LIN {X 0,Y 566.425,Z 352.194,A -85,B 0,C 180,E1 -2599.455,E2 -2599.455} C_VEL
LIN {X 0,Y 566.296,Z 363.628,A -85,B 0,C 180,E1 -2600.355,E2 -2600.355} C_VEL
LIN {X 0,Y 566.162,Z 372.742,A -85,B 0,C 180,E1 -2601.254,E2 -2601.254} C_VEL
LIN {X 0,Y 566.096,Z 380.288,A -85,B 0,C 180,E1 -2602.151,E2 -2602.151} C_VEL
LIN {X 0,Y 566.007,Z 386.693,A -85,B 0,C 180,E1 -2603.065,E2 -2603.065} C_VEL
LIN {X 0,Y 565.99,Z 391.812,A -85,B 0,C 180,E1 -2603.942,E2 -2603.942} C_VEL
LIN {X 0,Y 565.878,Z 396.909,A -85,B 0,C 180,E1 -2605.013,E2 -2605.013} C_VEL
LIN {X 0,Y 565.927,Z 400.862,A -85,B 0,C 180,E1 -2606.084,E2 -2606.084} C_VEL
LIN {X 0,Y 565.878,Z 403.78,A -85,B 0,C 180,E1 -2607.153,E2 -2607.153} C_VEL
LIN {X 0,Y 565.846,Z 406.194,A -85,B 0,C 180,E1 -2608.577,E2 -2608.577} C_VEL
LIN {X 0,Y 565.841,Z 406.781,A -85,B 0,C 180,E1 -2609.288,E2 -2609.288} C_VEL
LIN {X 0,Y 565.841,Z 406.781,A -85,B 0,C 180,E1 -2610.712,E2 -2610.712} C_VEL
LIN {X 0,Y 565.846,Z 406.194,A -85,B 0,C 180,E1 -2611.423,E2 -2611.423} C_VEL
LIN {X 0,Y 565.878,Z 403.78,A -85,B 0,C 180,E1 -2612.847,E2 -2612.847} C_VEL
LIN {X 0,Y 565.927,Z 400.862,A -85,B 0,C 180,E1 -2613.916,E2 -2613.916} C_VEL
LIN {X 0,Y 565.878,Z 396.909,A -85,B 0,C 180,E1 -2614.987,E2 -2614.987} C_VEL
LIN {X 0,Y 565.991,Z 391.812,A -85,B 0,C 180,E1 -2616.058,E2 -2616.058} C_VEL
LIN {X 0,Y 566.035,Z 385.428,A -85,B 0,C 180,E1 -2617.132,E2 -2617.132} C_VEL
LIN {X 0,Y 566.134,Z 377.5,A -85,B 0,C 180,E1 -2618.207,E2 -2618.207} C_VEL
LIN {X 0,Y 566.239,Z 369.359,A -85,B 0,C 180,E1 -2619.105,E2 -2619.105} C_VEL
LIN {X 0,Y 566.339,Z 359.324,A -85,B 0,C 180,E1 -2620.005,E2 -2620.005} C_VEL
LIN {X 0,Y 566.458,Z 349.496,A -85,B 0,C 180,E1 -2620.725,E2 -2620.725} C_VEL
LIN {X 0,Y 566.565,Z 338.733,A -85,B 0,C 180,E1 -2621.366,E2 -2621.366} C_VEL
LIN {X 0,Y 566.736,Z 324.932,A -85,B 0,C 180,E1 -2621.988,E2 -2621.988} C_VEL
LIN {X 0,Y 566.892,Z 312.891,A -85,B 0,C 180,E1 -2622.371,E2 -2622.371} C_VEL
LIN {X 0,Y 566.7,Z 306.442,A -85,B 0,C 180,E1 -2622.534,E2 -2622.534} C_VEL
LIN {X 0,Y 565.903,Z 301.524,A -85,B 0,C 180,E1 -2622.643,E2 -2622.643} C_VEL
LIN {X 0,Y 565.956,Z 295.461,A -85,B 0,C 180,E1 -2625.116,E2 -2625.116} C_VEL
LIN {X 0,Y 566.005,Z 288.275,A -85,B 0,C 180,E1 -2628.084,E2 -2628.084} C_VEL
LIN {X 0,Y 566.01,Z 282.873,A -85,B 0,C 180,E1 -2630.344,E2 -2630.344} C_VEL
LIN {X 0,Y 566.031,Z 277.383,A -85,B 0,C 180,E1 -2632.637,E2 -2632.637} C_VEL
LIN {X 0,Y 566.079,Z 272.028,A -85,B 0,C 180,E1 -2634.997,E2 -2634.997} C_VEL
LIN {X 0,Y 566.145,Z 266.834,A -85,B 0,C 180,E1 -2637.342,E2 -2637.342} C_VEL
LIN {X 0,Y 566.199,Z 261.606,A -85,B 0,C 180,E1 -2639.768,E2 -2639.768} C_VEL
LIN {X 0,Y 566.325,Z 256.131,A -85,B 0,C 180,E1 -2642.447,E2 -2642.447} C_VEL
LIN {X 0,Y 566.395,Z 249.901,A -85,B 0,C 180,E1 -2645.674,E2 -2645.674} C_VEL
LIN {X 0,Y 566.483,Z 244.633,A -85,B 0,C 180,E1 -2648.59,E2 -2648.59} C_VEL
LIN {X 0,Y 566.516,Z 240.41,A -85,B 0,C 180,E1 -2651.108,E2 -2651.108} C_VEL
LIN {X 0,Y 566.447,Z 237.397,A -85,B 0,C 180,E1 -2653.03,E2 -2653.03} C_VEL
LIN {X 0,Y 566.232,Z 235.917,A -85,B 0,C 180,E1 -2654.031,E2 -2654.031} C_VEL
LIN {X 0,Y 566.168,Z 235.461,A -85,B 0,C 180,E1 -2655.035,E2 -2655.035} C_VEL
LIN {X 0,Y 566.176,Z 235.461,A -85,B 0,C 180,E1 -2657.907,E2 -2657.907} C_VEL
LIN {X 0,Y 566.209,Z 235.454,A -85,B 0,C 180,E1 -2660.723,E2 -2660.723} C_VEL
LIN {X 0,Y 566.181,Z 235.456,A -85,B 0,C 180,E1 -2663.426,E2 -2663.426} C_VEL
LIN {X 0,Y 566.213,Z 235.456,A -85,B 0,C 180,E1 -2666.264,E2 -2666.264} C_VEL
LIN {X 0,Y 566.185,Z 235.453,A -85,B 0,C 180,E1 -2668.922,E2 -2668.922} C_VEL
LIN {X 0,Y 566.188,Z 235.461,A -85,B 0,C 180,E1 -2671.853,E2 -2671.853} C_VEL
LIN {X 0,Y 566.238,Z 235.447,A -85,B 0,C 180,E1 -2675.036,E2 -2675.036} C_VEL
LIN {X 0,Y 566.189,Z 235.457,A -85,B 0,C 180,E1 -2678.134,E2 -2678.134} C_VEL
LIN {X 0,Y 566.228,Z 235.448,A -85,B 0,C 180,E1 -2680.611,E2 -2680.611} C_VEL
LIN {X 0,Y 566.194,Z 235.458,A -85,B 0,C 180,E1 -2683.408,E2 -2683.408} C_VEL
LIN {X 0,Y 566.183,Z 235.454,A -85,B 0,C 180,E1 -2686.355,E2 -2686.355} C_VEL
LIN {X 0,Y 566.226,Z 235.454,A -85,B 0,C 180,E1 -2689.267,E2 -2689.267} C_VEL
LIN {X 0,Y 566.179,Z 235.455,A -85,B 0,C 180,E1 -2692.148,E2 -2692.148} C_VEL
LIN {X 0,Y 566.231,Z 235.447,A -85,B 0,C 180,E1 -2694.298,E2 -2694.298} C_VEL
LIN {X 0,Y 566.255,Z 235.452,A -85,B 0,C 180,E1 -2697.15,E2 -2697.15} C_VEL
LIN {X 0,Y 566.265,Z 235.444,A -85,B 0,C 180,E1 -2699.996,E2 -2699.996} C_VEL
LIN {X 0,Y 566.25,Z 235.45,A -85,B 0,C 180,E1 -2702.841,E2 -2702.841} C_VEL
LIN {X 0,Y 566.235,Z 235.448,A -85,B 0,C 180,E1 -2705.694,E2 -2705.694} C_VEL
LIN {X 0,Y 566.178,Z 235.457,A -85,B 0,C 180,E1 -2708.562,E2 -2708.562} C_VEL
LIN {X 0,Y 566.231,Z 235.45,A -85,B 0,C 180,E1 -2711.45,E2 -2711.45} C_VEL
LIN {X 0,Y 566.205,Z 235.454,A -85,B 0,C 180,E1 -2714.5,E2 -2714.5} C_VEL
LIN {X 0,Y 566.171,Z 235.457,A -85,B 0,C 180,E1 -2717.327,E2 -2717.327} C_VEL
LIN {X 0,Y 566.19,Z 235.456,A -85,B 0,C 180,E1 -2720.332,E2 -2720.332} C_VEL
LIN {X 0,Y 566.141,Z 235.46,A -85,B 0,C 180,E1 -2723.277,E2 -2723.277} C_VEL
LIN {X 0,Y 566.178,Z 235.454,A -85,B 0,C 180,E1 -2725.744,E2 -2725.744} C_VEL
LIN {X 0,Y 566.178,Z 235.454,A -85,B 0,C 180,E1 -2727.457,E2 -2727.457} C_VEL
LIN {X 0,Y 565.499,Z 235.542,A -85,B 0,C 180,E1 -2728.051,E2 -2728.051} C_VEL
LIN {X 0,Y 562.63,Z 235.898,A -85,B 0,C 180,E1 -2729.015,E2 -2729.015} C_VEL
LIN {X 0,Y 560.214,Z 236.2,A -85,B 0,C 180,E1 -2729.79,E2 -2729.79} C_VEL
LIN {X 0,Y 559.183,Z 236.334,A -85,B 0,C 180,E1 -2730.389,E2 -2730.389} C_VEL
LIN {X 0,Y 559.102,Z 236.337,A -85,B 0,C 180,E1 -2730.592,E2 -2730.592} C_VEL
LIN {X 0,Y 559.137,Z 236.331,A -85,B 0,C 180,E1 -2733.569,E2 -2733.569} C_VEL
LIN {X 0,Y 559.146,Z 236.338,A -85,B 0,C 180,E1 -2736.447,E2 -2736.447} C_VEL
LIN {X 0,Y 559.131,Z 236.333,A -85,B 0,C 180,E1 -2738.929,E2 -2738.929} C_VEL
LIN {X 0,Y 559.154,Z 236.332,A -85,B 0,C 180,E1 -2741.762,E2 -2741.762} C_VEL
LIN {X 0,Y 559.109,Z 236.336,A -85,B 0,C 180,E1 -2744.733,E2 -2744.733} C_VEL
LIN {X 0,Y 559.134,Z 236.338,A -85,B 0,C 180,E1 -2747.857,E2 -2747.857} C_VEL
LIN {X 0,Y 559.14,Z 236.338,A -85,B 0,C 180,E1 -2750.132,E2 -2750.132} C_VEL
LIN {X 0,Y 559.091,Z 236.337,A -85,B 0,C 180,E1 -2752.889,E2 -2752.889} C_VEL
LIN {X 0,Y 559.105,Z 236.34,A -85,B 0,C 180,E1 -2755.553,E2 -2755.553} C_VEL
LIN {X 0,Y 559.118,Z 236.338,A -85,B 0,C 180,E1 -2758.135,E2 -2758.135} C_VEL
LIN {X 0,Y 559.12,Z 236.333,A -85,B 0,C 180,E1 -2760.646,E2 -2760.646} C_VEL
LIN {X 0,Y 559.12,Z 236.336,A -85,B 0,C 180,E1 -2763.167,E2 -2763.167} C_VEL
LIN {X 0,Y 559.11,Z 236.342,A -85,B 0,C 180,E1 -2765.493,E2 -2765.493} C_VEL
LIN {X 0,Y 559.104,Z 236.34,A -85,B 0,C 180,E1 -2767.846,E2 -2767.846} C_VEL
LIN {X 0,Y 559.131,Z 236.332,A -85,B 0,C 180,E1 -2770.49,E2 -2770.49} C_VEL
LIN {X 0,Y 559.146,Z 236.337,A -85,B 0,C 180,E1 -2773.197,E2 -2773.197} C_VEL
LIN {X 0,Y 559.12,Z 236.334,A -85,B 0,C 180,E1 -2776.183,E2 -2776.183} C_VEL
LIN {X 0,Y 559.171,Z 236.335,A -85,B 0,C 180,E1 -2779.133,E2 -2779.133} C_VEL
LIN {X 0,Y 559.149,Z 236.331,A -85,B 0,C 180,E1 -2782.053,E2 -2782.053} C_VEL
LIN {X 0,Y 559.203,Z 236.331,A -85,B 0,C 180,E1 -2784.953,E2 -2784.953} C_VEL
LIN {X 0,Y 559.183,Z 236.327,A -85,B 0,C 180,E1 -2787.839,E2 -2787.839} C_VEL
LIN {X 0,Y 559.219,Z 236.328,A -85,B 0,C 180,E1 -2790.72,E2 -2790.72} C_VEL
LIN {X 0,Y 559.187,Z 236.334,A -85,B 0,C 180,E1 -2792.882,E2 -2792.882} C_VEL
LIN {X 0,Y 559.173,Z 236.328,A -85,B 0,C 180,E1 -2795.771,E2 -2795.771} C_VEL
LIN {X 0,Y 559.149,Z 236.331,A -85,B 0,C 180,E1 -2797.947,E2 -2797.947} C_VEL
LIN {X 0,Y 559.171,Z 236.335,A -85,B 0,C 180,E1 -2800.867,E2 -2800.867} C_VEL
LIN {X 0,Y 559.12,Z 236.334,A -85,B 0,C 180,E1 -2803.817,E2 -2803.817} C_VEL
LIN {X 0,Y 559.146,Z 236.337,A -85,B 0,C 180,E1 -2806.803,E2 -2806.803} C_VEL
LIN {X 0,Y 559.113,Z 236.335,A -85,B 0,C 180,E1 -2809.839,E2 -2809.839} C_VEL
LIN {X 0,Y 559.103,Z 236.34,A -85,B 0,C 180,E1 -2812.154,E2 -2812.154} C_VEL
LIN {X 0,Y 559.11,Z 236.342,A -85,B 0,C 180,E1 -2814.507,E2 -2814.507} C_VEL
LIN {X 0,Y 559.118,Z 236.335,A -85,B 0,C 180,E1 -2816.904,E2 -2816.904} C_VEL
LIN {X 0,Y 559.141,Z 236.334,A -85,B 0,C 180,E1 -2819.871,E2 -2819.871} C_VEL
LIN {X 0,Y 559.118,Z 236.336,A -85,B 0,C 180,E1 -2822.717,E2 -2822.717} C_VEL
LIN {X 0,Y 559.101,Z 236.336,A -85,B 0,C 180,E1 -2825.325,E2 -2825.325} C_VEL
LIN {X 0,Y 559.09,Z 236.346,A -85,B 0,C 180,E1 -2828.02,E2 -2828.02} C_VEL
LIN {X 0,Y 559.125,Z 236.333,A -85,B 0,C 180,E1 -2830.814,E2 -2830.814} C_VEL
LIN {X 0,Y 559.111,Z 236.341,A -85,B 0,C 180,E1 -2833.736,E2 -2833.736} C_VEL
LIN {X 0,Y 559.129,Z 236.332,A -85,B 0,C 180,E1 -2836.804,E2 -2836.804} C_VEL
LIN {X 0,Y 559.132,Z 236.333,A -85,B 0,C 180,E1 -2839.194,E2 -2839.194} C_VEL
LIN {X 0,Y 559.09,Z 236.342,A -85,B 0,C 180,E1 -2841.987,E2 -2841.987} C_VEL
LIN {X 0,Y 559.116,Z 236.334,A -85,B 0,C 180,E1 -2844.683,E2 -2844.683} C_VEL
LIN {X 0,Y 559.135,Z 236.337,A -85,B 0,C 180,E1 -2847.366,E2 -2847.366} C_VEL
LIN {X 0,Y 559.111,Z 236.335,A -85,B 0,C 180,E1 -2850.147,E2 -2850.147} C_VEL
LIN {X 0,Y 559.136,Z 236.336,A -85,B 0,C 180,E1 -2853.102,E2 -2853.102} C_VEL
LIN {X 0,Y 559.124,Z 236.34,A -85,B 0,C 180,E1 -2855.5,E2 -2855.5} C_VEL
LIN {X 0,Y 559.147,Z 236.331,A -85,B 0,C 180,E1 -2858.629,E2 -2858.629} C_VEL
LIN {X 0,Y 559.14,Z 236.335,A -85,B 0,C 180,E1 -2860.931,E2 -2860.931} C_VEL
LIN {X 0,Y 559.139,Z 236.331,A -85,B 0,C 180,E1 -2863.952,E2 -2863.952} C_VEL
LIN {X 0,Y 559.144,Z 236.33,A -85,B 0,C 180,E1 -2866.189,E2 -2866.189} C_VEL
LIN {X 0,Y 559.186,Z 236.333,A -85,B 0,C 180,E1 -2869.138,E2 -2869.138} C_VEL
LIN {X 0,Y 559.173,Z 236.327,A -85,B 0,C 180,E1 -2872.058,E2 -2872.058} C_VEL
LIN {X 0,Y 559.231,Z 236.328,A -85,B 0,C 180,E1 -2874.958,E2 -2874.958} C_VEL
LIN {X 0,Y 559.223,Z 236.32,A -85,B 0,C 180,E1 -2877.844,E2 -2877.844} C_VEL
LIN {X 0,Y 559.267,Z 236.324,A -85,B 0,C 180,E1 -2880.724,E2 -2880.724} C_VEL
LIN {X 0,Y 559.22,Z 236.327,A -85,B 0,C 180,E1 -2882.886,E2 -2882.886} C_VEL
LIN {X 0,Y 559.202,Z 236.323,A -85,B 0,C 180,E1 -2885.774,E2 -2885.774} C_VEL
LIN {X 0,Y 559.154,Z 236.336,A -85,B 0,C 180,E1 -2888.679,E2 -2888.679} C_VEL
LIN {X 0,Y 559.196,Z 236.324,A -85,B 0,C 180,E1 -2891.604,E2 -2891.604} C_VEL
LIN {X 0,Y 559.197,Z 236.33,A -85,B 0,C 180,E1 -2894.599,E2 -2894.599} C_VEL
LIN {X 0,Y 559.129,Z 236.332,A -85,B 0,C 180,E1 -2897.561,E2 -2897.561} C_VEL
LIN {X 0,Y 559.161,Z 236.331,A -85,B 0,C 180,E1 -2899.841,E2 -2899.841} C_VEL
LIN {X 0,Y 559.137,Z 236.34,A -85,B 0,C 180,E1 -2902.156,E2 -2902.156} C_VEL
LIN {X 0,Y 559.154,Z 236.329,A -85,B 0,C 180,E1 -2905.302,E2 -2905.302} C_VEL
LIN {X 0,Y 559.128,Z 236.335,A -85,B 0,C 180,E1 -2908.534,E2 -2908.534} C_VEL
LIN {X 0,Y 559.142,Z 236.331,A -85,B 0,C 180,E1 -2911.275,E2 -2911.275} C_VEL
LIN {X 0,Y 559.166,Z 236.337,A -85,B 0,C 180,E1 -2913.951,E2 -2913.951} C_VEL
LIN {X 0,Y 559.131,Z 236.334,A -85,B 0,C 180,E1 -2917.112,E2 -2917.112} C_VEL
LIN {X 0,Y 559.16,Z 236.337,A -85,B 0,C 180,E1 -2919.943,E2 -2919.943} C_VEL
LIN {X 0,Y 559.149,Z 236.333,A -85,B 0,C 180,E1 -2922.747,E2 -2922.747} C_VEL
LIN {X 0,Y 559.128,Z 236.342,A -85,B 0,C 180,E1 -2925.261,E2 -2925.261} C_VEL
LIN {X 0,Y 559.491,Z 239.126,A -85,B 0,C 180,E1 -2927.289,E2 -2927.289} C_VEL
LIN {X 0,Y 559.518,Z 243.446,A -85,B 0,C 180,E1 -2930.017,E2 -2930.017} C_VEL
LIN {X 0,Y 559.416,Z 248.448,A -85,B 0,C 180,E1 -2932.914,E2 -2932.914} C_VEL
LIN {X 0,Y 559.316,Z 253.303,A -85,B 0,C 180,E1 -2935.568,E2 -2935.568} C_VEL
LIN {X 0,Y 559.244,Z 258.304,A -85,B 0,C 180,E1 -2938.143,E2 -2938.143} C_VEL
LIN {X 0,Y 559.118,Z 263.414,A -85,B 0,C 180,E1 -2940.646,E2 -2940.646} C_VEL
LIN {X 0,Y 559.095,Z 268.793,A -85,B 0,C 180,E1 -2943.19,E2 -2943.19} C_VEL
LIN {X 0,Y 558.976,Z 275.599,A -85,B 0,C 180,E1 -2946.276,E2 -2946.276} C_VEL
LIN {X 0,Y 558.99,Z 280.952,A -85,B 0,C 180,E1 -2948.617,E2 -2948.617} C_VEL
LIN {X 0,Y 558.923,Z 288.261,A -85,B 0,C 180,E1 -2951.679,E2 -2951.679} C_VEL
LIN {X 0,Y 558.869,Z 295.461,A -85,B 0,C 180,E1 -2954.688,E2 -2954.688} C_VEL
LIN {X 0,Y 558.838,Z 301.524,A -85,B 0,C 180,E1 -2957.194,E2 -2957.194} C_VEL
LIN {X 0,Y 559.997,Z 310.238,A -85,B 0,C 180,E1 -2957.405,E2 -2957.405} C_VEL
LIN {X 0,Y 559.848,Z 321.177,A -85,B 0,C 180,E1 -2957.729,E2 -2957.729} C_VEL
LIN {X 0,Y 559.718,Z 330.187,A -85,B 0,C 180,E1 -2958.08,E2 -2958.08} C_VEL
LIN {X 0,Y 559.585,Z 340.522,A -85,B 0,C 180,E1 -2958.592,E2 -2958.592} C_VEL
LIN {X 0,Y 559.46,Z 350.83,A -85,B 0,C 180,E1 -2959.231,E2 -2959.231} C_VEL
LIN {X 0,Y 559.317,Z 360.442,A -85,B 0,C 180,E1 -2959.96,E2 -2959.96} C_VEL
LIN {X 0,Y 559.197,Z 371.11,A -85,B 0,C 180,E1 -2960.962,E2 -2960.962} C_VEL
LIN {X 0,Y 559.051,Z 378.909,A -85,B 0,C 180,E1 -2961.87,E2 -2961.87} C_VEL
LIN {X 0,Y 558.977,Z 385.419,A -85,B 0,C 180,E1 -2962.777,E2 -2962.777} C_VEL
LIN {X 0,Y 558.91,Z 391.803,A -85,B 0,C 180,E1 -2963.864,E2 -2963.864} C_VEL
LIN {X 0,Y 558.798,Z 396.9,A -85,B 0,C 180,E1 -2964.949,E2 -2964.949} C_VEL
LIN {X 0,Y 558.845,Z 400.855,A -85,B 0,C 180,E1 -2966.034,E2 -2966.034} C_VEL
LIN {X 0,Y 558.8,Z 403.775,A -85,B 0,C 180,E1 -2967.116,E2 -2967.116} C_VEL
LIN {X 0,Y 558.745,Z 406.195,A -85,B 0,C 180,E1 -2968.559,E2 -2968.559} C_VEL
LIN {X 0,Y 558.741,Z 406.78,A -85,B 0,C 180,E1 -2969.279,E2 -2969.279} C_VEL
LIN {X 0,Y 558.741,Z 406.78,A -85,B 0,C 180,E1 -2970.721,E2 -2970.721} C_VEL
LIN {X 0,Y 558.745,Z 406.195,A -85,B 0,C 180,E1 -2971.441,E2 -2971.441} C_VEL
LIN {X 0,Y 558.8,Z 403.775,A -85,B 0,C 180,E1 -2972.884,E2 -2972.884} C_VEL
LIN {X 0,Y 558.845,Z 400.855,A -85,B 0,C 180,E1 -2973.966,E2 -2973.966} C_VEL
LIN {X 0,Y 558.798,Z 396.9,A -85,B 0,C 180,E1 -2975.051,E2 -2975.051} C_VEL
LIN {X 0,Y 558.911,Z 391.803,A -85,B 0,C 180,E1 -2976.136,E2 -2976.136} C_VEL
LIN {X 0,Y 558.977,Z 385.419,A -85,B 0,C 180,E1 -2977.223,E2 -2977.223} C_VEL
LIN {X 0,Y 559.098,Z 377.503,A -85,B 0,C 180,E1 -2978.311,E2 -2978.311} C_VEL
LIN {X 0,Y 559.212,Z 369.36,A -85,B 0,C 180,E1 -2979.22,E2 -2979.22} C_VEL
LIN {X 0,Y 559.349,Z 359.311,A -85,B 0,C 180,E1 -2980.131,E2 -2980.131} C_VEL
LIN {X 0,Y 559.46,Z 350.83,A -85,B 0,C 180,E1 -2980.769,E2 -2980.769} C_VEL
LIN {X 0,Y 559.578,Z 340.587,A -85,B 0,C 180,E1 -2981.404,E2 -2981.404} C_VEL
LIN {X 0,Y 559.729,Z 330.496,A -85,B 0,C 180,E1 -2981.906,E2 -2981.906} C_VEL
LIN {X 0,Y 559.875,Z 319.762,A -85,B 0,C 180,E1 -2982.321,E2 -2982.321} C_VEL
LIN {X 0,Y 559.823,Z 307.537,A -85,B 0,C 180,E1 -2982.668,E2 -2982.668} C_VEL
LIN {X 0,Y 558.839,Z 301.524,A -85,B 0,C 180,E1 -2982.806,E2 -2982.806} C_VEL
LIN {X 0,Y 558.869,Z 295.461,A -85,B 0,C 180,E1 -2985.312,E2 -2985.312} C_VEL
LIN {X 0,Y 558.923,Z 288.261,A -85,B 0,C 180,E1 -2988.321,E2 -2988.321} C_VEL
LIN {X 0,Y 558.99,Z 280.952,A -85,B 0,C 180,E1 -2991.383,E2 -2991.383} C_VEL
LIN {X 0,Y 558.998,Z 273.846,A -85,B 0,C 180,E1 -2994.512,E2 -2994.512} C_VEL
LIN {X 0,Y 559.077,Z 268.585,A -85,B 0,C 180,E1 -2996.906,E2 -2996.906} C_VEL
LIN {X 0,Y 559.17,Z 262.314,A -85,B 0,C 180,E1 -2999.859,E2 -2999.859} C_VEL
LIN {X 0,Y 559.281,Z 256.61,A -85,B 0,C 180,E1 -3002.706,E2 -3002.706} C_VEL
LIN {X 0,Y 559.387,Z 251.651,A -85,B 0,C 180,E1 -3005.304,E2 -3005.304} C_VEL
LIN {X 0,Y 559.435,Z 246.829,A -85,B 0,C 180,E1 -3007.992,E2 -3007.992} C_VEL
LIN {X 0,Y 559.522,Z 242.141,A -85,B 0,C 180,E1 -3010.779,E2 -3010.779} C_VEL
LIN {X 0,Y 559.411,Z 238.339,A -85,B 0,C 180,E1 -3013.223,E2 -3013.223} C_VEL
LIN {X 0,Y 559.125,Z 236.341,A -85,B 0,C 180,E1 -3014.739,E2 -3014.739} C_VEL
LIN {X 0,Y 559.144,Z 236.337,A -85,B 0,C 180,E1 -3017.865,E2 -3017.865} C_VEL
LIN {X 0,Y 559.178,Z 236.335,A -85,B 0,C 180,E1 -3020.132,E2 -3020.132} C_VEL
LIN {X 0,Y 559.131,Z 236.334,A -85,B 0,C 180,E1 -3022.888,E2 -3022.888} C_VEL
LIN {X 0,Y 559.166,Z 236.337,A -85,B 0,C 180,E1 -3026.049,E2 -3026.049} C_VEL
LIN {X 0,Y 559.15,Z 236.329,A -85,B 0,C 180,E1 -3028.978,E2 -3028.978} C_VEL
LIN {X 0,Y 559.134,Z 236.336,A -85,B 0,C 180,E1 -3031.623,E2 -3031.623} C_VEL
LIN {X 0,Y 559.161,Z 236.328,A -85,B 0,C 180,E1 -3034.814,E2 -3034.814} C_VEL
LIN {X 0,Y 559.137,Z 236.34,A -85,B 0,C 180,E1 -3037.844,E2 -3037.844} C_VEL
LIN {X 0,Y 559.19,Z 236.325,A -85,B 0,C 180,E1 -3040.491,E2 -3040.491} C_VEL
LIN {X 0,Y 559.162,Z 236.331,A -85,B 0,C 180,E1 -3043.194,E2 -3043.194} C_VEL
LIN {X 0,Y 559.16,Z 236.33,A -85,B 0,C 180,E1 -3046.18,E2 -3046.18} C_VEL
LIN {X 0,Y 559.184,Z 236.329,A -85,B 0,C 180,E1 -3049.13,E2 -3049.13} C_VEL
LIN {X 0,Y 559.133,Z 236.333,A -85,B 0,C 180,E1 -3052.049,E2 -3052.049} C_VEL
LIN {X 0,Y 559.202,Z 236.323,A -85,B 0,C 180,E1 -3054.226,E2 -3054.226} C_VEL
LIN {X 0,Y 559.22,Z 236.327,A -85,B 0,C 180,E1 -3057.114,E2 -3057.114} C_VEL
LIN {X 0,Y 559.237,Z 236.319,A -85,B 0,C 180,E1 -3059.996,E2 -3059.996} C_VEL
LIN {X 0,Y 559.218,Z 236.326,A -85,B 0,C 180,E1 -3062.877,E2 -3062.877} C_VEL
LIN {X 0,Y 559.202,Z 236.324,A -85,B 0,C 180,E1 -3065.766,E2 -3065.766} C_VEL
LIN {X 0,Y 559.144,Z 236.334,A -85,B 0,C 180,E1 -3068.67,E2 -3068.67} C_VEL
LIN {X 0,Y 559.188,Z 236.326,A -85,B 0,C 180,E1 -3071.596,E2 -3071.596} C_VEL
LIN {X 0,Y 559.176,Z 236.331,A -85,B 0,C 180,E1 -3074.591,E2 -3074.591} C_VEL
LIN {X 0,Y 559.115,Z 236.334,A -85,B 0,C 180,E1 -3077.553,E2 -3077.553} C_VEL
LIN {X 0,Y 559.146,Z 236.33,A -85,B 0,C 180,E1 -3079.833,E2 -3079.833} C_VEL
LIN {X 0,Y 559.111,Z 236.336,A -85,B 0,C 180,E1 -3082.148,E2 -3082.148} C_VEL
LIN {X 0,Y 559.142,Z 236.331,A -85,B 0,C 180,E1 -3085.293,E2 -3085.293} C_VEL
LIN {X 0,Y 559.137,Z 236.338,A -85,B 0,C 180,E1 -3088.378,E2 -3088.378} C_VEL
LIN {X 0,Y 559.102,Z 236.337,A -85,B 0,C 180,E1 -3090.592,E2 -3090.592} C_VEL
LIN {X 0,Y 558.44,Z 236.42,A -85,B 0,C 180,E1 -3091.193,E2 -3091.193} C_VEL
LIN {X 0,Y 555.583,Z 236.779,A -85,B 0,C 180,E1 -3092.169,E2 -3092.169} C_VEL
LIN {X 0,Y 553.175,Z 237.076,A -85,B 0,C 180,E1 -3092.955,E2 -3092.955} C_VEL
LIN {X 0,Y 552.156,Z 237.201,A -85,B 0,C 180,E1 -3093.562,E2 -3093.562} C_VEL
LIN {X 0,Y 552.082,Z 237.211,A -85,B 0,C 180,E1 -3093.767,E2 -3093.767} C_VEL
LIN {X 0,Y 552.074,Z 237.214,A -85,B 0,C 180,E1 -3096.742,E2 -3096.742} C_VEL
LIN {X 0,Y 552.088,Z 237.21,A -85,B 0,C 180,E1 -3099.522,E2 -3099.522} C_VEL
LIN {X 0,Y 552.124,Z 237.205,A -85,B 0,C 180,E1 -3101.437,E2 -3101.437} C_VEL
LIN {X 0,Y 552.067,Z 237.215,A -85,B 0,C 180,E1 -3104.53,E2 -3104.53} C_VEL
LIN {X 0,Y 552.078,Z 237.213,A -85,B 0,C 180,E1 -3107.58,E2 -3107.58} C_VEL
LIN {X 0,Y 552.102,Z 237.21,A -85,B 0,C 180,E1 -3110.472,E2 -3110.472} C_VEL
LIN {X 0,Y 552.057,Z 237.215,A -85,B 0,C 180,E1 -3113.312,E2 -3113.312} C_VEL
LIN {X 0,Y 552.082,Z 237.218,A -85,B 0,C 180,E1 -3115.937,E2 -3115.937} C_VEL
LIN {X 0,Y 552.057,Z 237.214,A -85,B 0,C 180,E1 -3118.537,E2 -3118.537} C_VEL
LIN {X 0,Y 552.083,Z 237.215,A -85,B 0,C 180,E1 -3121.431,E2 -3121.431} C_VEL
LIN {X 0,Y 552.11,Z 237.207,A -85,B 0,C 180,E1 -3124.355,E2 -3124.355} C_VEL
LIN {X 0,Y 552.092,Z 237.209,A -85,B 0,C 180,E1 -3126.758,E2 -3126.758} C_VEL
LIN {X 0,Y 552.072,Z 237.215,A -85,B 0,C 180,E1 -3129.897,E2 -3129.897} C_VEL
LIN {X 0,Y 552.125,Z 237.209,A -85,B 0,C 180,E1 -3132.977,E2 -3132.977} C_VEL
LIN {X 0,Y 552.078,Z 237.213,A -85,B 0,C 180,E1 -3136.003,E2 -3136.003} C_VEL
LIN {X 0,Y 552.129,Z 237.21,A -85,B 0,C 180,E1 -3138.993,E2 -3138.993} C_VEL
LIN {X 0,Y 552.103,Z 237.209,A -85,B 0,C 180,E1 -3141.951,E2 -3141.951} C_VEL
LIN {X 0,Y 552.143,Z 237.204,A -85,B 0,C 180,E1 -3144.156,E2 -3144.156} C_VEL
LIN {X 0,Y 552.153,Z 237.21,A -85,B 0,C 180,E1 -3147.082,E2 -3147.082} C_VEL
LIN {X 0,Y 552.158,Z 237.202,A -85,B 0,C 180,E1 -3150,E2 -3150} C_VEL
LIN {X 0,Y 552.153,Z 237.21,A -85,B 0,C 180,E1 -3152.918,E2 -3152.918} C_VEL
LIN {X 0,Y 552.143,Z 237.204,A -85,B 0,C 180,E1 -3155.844,E2 -3155.844} C_VEL
LIN {X 0,Y 552.103,Z 237.209,A -85,B 0,C 180,E1 -3158.049,E2 -3158.049} C_VEL
LIN {X 0,Y 552.129,Z 237.21,A -85,B 0,C 180,E1 -3161.007,E2 -3161.007} C_VEL
LIN {X 0,Y 552.078,Z 237.213,A -85,B 0,C 180,E1 -3163.997,E2 -3163.997} C_VEL
LIN {X 0,Y 552.126,Z 237.206,A -85,B 0,C 180,E1 -3167.343,E2 -3167.343} C_VEL
LIN {X 0,Y 552.072,Z 237.215,A -85,B 0,C 180,E1 -3170.103,E2 -3170.103} C_VEL
LIN {X 0,Y 552.092,Z 237.209,A -85,B 0,C 180,E1 -3173.242,E2 -3173.242} C_VEL
LIN {X 0,Y 552.11,Z 237.207,A -85,B 0,C 180,E1 -3175.645,E2 -3175.645} C_VEL
LIN {X 0,Y 552.083,Z 237.215,A -85,B 0,C 180,E1 -3178.569,E2 -3178.569} C_VEL
LIN {X 0,Y 552.074,Z 237.212,A -85,B 0,C 180,E1 -3181.483,E2 -3181.483} C_VEL
LIN {X 0,Y 552.088,Z 237.219,A -85,B 0,C 180,E1 -3184.176,E2 -3184.176} C_VEL
LIN {X 0,Y 552.055,Z 237.214,A -85,B 0,C 180,E1 -3186.75,E2 -3186.75} C_VEL
LIN {X 0,Y 552.114,Z 237.208,A -85,B 0,C 180,E1 -3189.527,E2 -3189.527} C_VEL
LIN {X 0,Y 552.078,Z 237.213,A -85,B 0,C 180,E1 -3192.429,E2 -3192.429} C_VEL
LIN {X 0,Y 552.071,Z 237.216,A -85,B 0,C 180,E1 -3195.569,E2 -3195.569} C_VEL
LIN {X 0,Y 552.124,Z 237.205,A -85,B 0,C 180,E1 -3198.677,E2 -3198.677} C_VEL
LIN {X 0,Y 552.074,Z 237.216,A -85,B 0,C 180,E1 -3201.416,E2 -3201.416} C_VEL
LIN {X 0,Y 552.07,Z 237.214,A -85,B 0,C 180,E1 -3204.163,E2 -3204.163} C_VEL
LIN {X 0,Y 552.089,Z 237.209,A -85,B 0,C 180,E1 -3206.82,E2 -3206.82} C_VEL
LIN {X 0,Y 552.065,Z 237.22,A -85,B 0,C 180,E1 -3209.395,E2 -3209.395} C_VEL
LIN {X 0,Y 552.091,Z 237.212,A -85,B 0,C 180,E1 -3211.907,E2 -3211.907} C_VEL
LIN {X 0,Y 552.122,Z 237.206,A -85,B 0,C 180,E1 -3214.654,E2 -3214.654} C_VEL
LIN {X 0,Y 552.062,Z 237.218,A -85,B 0,C 180,E1 -3217.554,E2 -3217.554} C_VEL
LIN {X 0,Y 552.122,Z 237.205,A -85,B 0,C 180,E1 -3220.378,E2 -3220.378} C_VEL
LIN {X 0,Y 552.129,Z 237.21,A -85,B 0,C 180,E1 -3222.982,E2 -3222.982} C_VEL
LIN {X 0,Y 552.109,Z 237.207,A -85,B 0,C 180,E1 -3226.009,E2 -3226.009} C_VEL
LIN {X 0,Y 552.155,Z 237.21,A -85,B 0,C 180,E1 -3228.998,E2 -3228.998} C_VEL
LIN {X 0,Y 552.128,Z 237.204,A -85,B 0,C 180,E1 -3231.956,E2 -3231.956} C_VEL
LIN {X 0,Y 552.206,Z 237.204,A -85,B 0,C 180,E1 -3234.893,E2 -3234.893} C_VEL
LIN {X 0,Y 552.197,Z 237.196,A -85,B 0,C 180,E1 -3237.816,E2 -3237.816} C_VEL
LIN {X 0,Y 552.236,Z 237.2,A -85,B 0,C 180,E1 -3240.733,E2 -3240.733} C_VEL
LIN {X 0,Y 552.185,Z 237.203,A -85,B 0,C 180,E1 -3242.922,E2 -3242.922} C_VEL
LIN {X 0,Y 552.175,Z 237.199,A -85,B 0,C 180,E1 -3245.848,E2 -3245.848} C_VEL
LIN {X 0,Y 552.127,Z 237.21,A -85,B 0,C 180,E1 -3248.79,E2 -3248.79} C_VEL
LIN {X 0,Y 552.152,Z 237.202,A -85,B 0,C 180,E1 -3251.754,E2 -3251.754} C_VEL
LIN {X 0,Y 552.132,Z 237.208,A -85,B 0,C 180,E1 -3254.752,E2 -3254.752} C_VEL
LIN {X 0,Y 552.088,Z 237.211,A -85,B 0,C 180,E1 -3257.793,E2 -3257.793} C_VEL
LIN {X 0,Y 552.122,Z 237.212,A -85,B 0,C 180,E1 -3260.105,E2 -3260.105} C_VEL
LIN {X 0,Y 552.088,Z 237.215,A -85,B 0,C 180,E1 -3262.454,E2 -3262.454} C_VEL
LIN {X 0,Y 552.121,Z 237.205,A -85,B 0,C 180,E1 -3265.346,E2 -3265.346} C_VEL
LIN {X 0,Y 552.095,Z 237.211,A -85,B 0,C 180,E1 -3268.559,E2 -3268.559} C_VEL
LIN {X 0,Y 552.114,Z 237.208,A -85,B 0,C 180,E1 -3271.478,E2 -3271.478} C_VEL
LIN {X 0,Y 552.107,Z 237.213,A -85,B 0,C 180,E1 -3274.168,E2 -3274.168} C_VEL
LIN {X 0,Y 552.1,Z 237.209,A -85,B 0,C 180,E1 -3276.75,E2 -3276.75} C_VEL
LIN {X 0,Y 552.129,Z 237.212,A -85,B 0,C 180,E1 -3279.53,E2 -3279.53} C_VEL
LIN {X 0,Y 552.112,Z 237.211,A -85,B 0,C 180,E1 -3282.43,E2 -3282.43} C_VEL
LIN {X 0,Y 552.085,Z 237.216,A -85,B 0,C 180,E1 -3284.532,E2 -3284.532} C_VEL
LIN {X 0,Y 552.165,Z 237.846,A -85,B 0,C 180,E1 -3285.571,E2 -3285.571} C_VEL
LIN {X 0,Y 552.511,Z 240.819,A -85,B 0,C 180,E1 -3287.612,E2 -3287.612} C_VEL
LIN {X 0,Y 552.485,Z 245.424,A -85,B 0,C 180,E1 -3290.504,E2 -3290.504} C_VEL
LIN {X 0,Y 552.408,Z 250.167,A -85,B 0,C 180,E1 -3293.277,E2 -3293.277} C_VEL
LIN {X 0,Y 552.289,Z 255.054,A -85,B 0,C 180,E1 -3295.951,E2 -3295.951} C_VEL
LIN {X 0,Y 552.164,Z 260.043,A -85,B 0,C 180,E1 -3298.544,E2 -3298.544} C_VEL
LIN {X 0,Y 552.074,Z 265.941,A -85,B 0,C 180,E1 -3301.45,E2 -3301.45} C_VEL
LIN {X 0,Y 551.961,Z 272.09,A -85,B 0,C 180,E1 -3304.348,E2 -3304.348} C_VEL
LIN {X 0,Y 551.907,Z 277.35,A -85,B 0,C 180,E1 -3306.75,E2 -3306.75} C_VEL
LIN {X 0,Y 551.865,Z 282.689,A -85,B 0,C 180,E1 -3309.11,E2 -3309.11} C_VEL
LIN {X 0,Y 551.839,Z 288.17,A -85,B 0,C 180,E1 -3311.435,E2 -3311.435} C_VEL
LIN {X 0,Y 551.784,Z 293.639,A -85,B 0,C 180,E1 -3313.728,E2 -3313.728} C_VEL
LIN {X 0,Y 551.762,Z 299.054,A -85,B 0,C 180,E1 -3315.995,E2 -3315.995} C_VEL
LIN {X 0,Y 551.736,Z 301.524,A -85,B 0,C 180,E1 -3317.026,E2 -3317.026} C_VEL
LIN {X 0,Y 553.043,Z 310.206,A -85,B 0,C 180,E1 -3317.244,E2 -3317.244} C_VEL
LIN {X 0,Y 552.926,Z 321.029,A -85,B 0,C 180,E1 -3317.568,E2 -3317.568} C_VEL
LIN {X 0,Y 552.752,Z 331.375,A -85,B 0,C 180,E1 -3317.983,E2 -3317.983} C_VEL
LIN {X 0,Y 552.595,Z 341.456,A -85,B 0,C 180,E1 -3318.5,E2 -3318.5} C_VEL
LIN {X 0,Y 552.47,Z 350.814,A -85,B 0,C 180,E1 -3319.093,E2 -3319.093} C_VEL
LIN {X 0,Y 552.301,Z 360.43,A -85,B 0,C 180,E1 -3319.831,E2 -3319.831} C_VEL
LIN {X 0,Y 552.152,Z 371.103,A -85,B 0,C 180,E1 -3320.845,E2 -3320.845} C_VEL
LIN {X 0,Y 552.014,Z 378.901,A -85,B 0,C 180,E1 -3321.765,E2 -3321.765} C_VEL
LIN {X 0,Y 551.907,Z 385.41,A -85,B 0,C 180,E1 -3322.684,E2 -3322.684} C_VEL
LIN {X 0,Y 551.812,Z 391.107,A -85,B 0,C 180,E1 -3323.653,E2 -3323.653} C_VEL
LIN {X 0,Y 551.803,Z 395.348,A -85,B 0,C 180,E1 -3324.519,E2 -3324.519} C_VEL
LIN {X 0,Y 551.767,Z 399.64,A -85,B 0,C 180,E1 -3325.617,E2 -3325.617} C_VEL
LIN {X 0,Y 551.751,Z 401.976,A -85,B 0,C 180,E1 -3326.349,E2 -3326.349} C_VEL
LIN {X 0,Y 551.724,Z 403.77,A -85,B 0,C 180,E1 -3327.079,E2 -3327.079} C_VEL
LIN {X 0,Y 551.645,Z 406.195,A -85,B 0,C 180,E1 -3328.54,E2 -3328.54} C_VEL
LIN {X 0,Y 551.641,Z 406.78,A -85,B 0,C 180,E1 -3329.27,E2 -3329.27} C_VEL
LIN {X 0,Y 551.641,Z 406.78,A -85,B 0,C 180,E1 -3330.73,E2 -3330.73} C_VEL
LIN {X 0,Y 551.645,Z 406.195,A -85,B 0,C 180,E1 -3331.46,E2 -3331.46} C_VEL
LIN {X 0,Y 551.724,Z 403.77,A -85,B 0,C 180,E1 -3332.921,E2 -3332.921} C_VEL
LIN {X 0,Y 551.765,Z 400.848,A -85,B 0,C 180,E1 -3334.017,E2 -3334.017} C_VEL
LIN {X 0,Y 551.724,Z 396.892,A -85,B 0,C 180,E1 -3335.116,E2 -3335.116} C_VEL
LIN {X 0,Y 551.838,Z 392.402,A -85,B 0,C 180,E1 -3336.097,E2 -3336.097} C_VEL
LIN {X 0,Y 551.89,Z 386.56,A -85,B 0,C 180,E1 -3337.132,E2 -3337.132} C_VEL
LIN {X 0,Y 551.986,Z 380.271,A -85,B 0,C 180,E1 -3338.051,E2 -3338.051} C_VEL
LIN {X 0,Y 552.124,Z 372.725,A -85,B 0,C 180,E1 -3338.971,E2 -3338.971} C_VEL
LIN {X 0,Y 552.274,Z 363.618,A -85,B 0,C 180,E1 -3339.892,E2 -3339.892} C_VEL
LIN {X 0,Y 552.45,Z 352.163,A -85,B 0,C 180,E1 -3340.815,E2 -3340.815} C_VEL
LIN {X 0,Y 552.571,Z 343.467,A -85,B 0,C 180,E1 -3341.386,E2 -3341.386} C_VEL
LIN {X 0,Y 552.745,Z 333.386,A -85,B 0,C 180,E1 -3341.924,E2 -3341.924} C_VEL
LIN {X 0,Y 552.892,Z 323.602,A -85,B 0,C 180,E1 -3342.34,E2 -3342.34} C_VEL
LIN {X 0,Y 553.04,Z 312.827,A -85,B 0,C 180,E1 -3342.686,E2 -3342.686} C_VEL
LIN {X 0,Y 552.767,Z 307.533,A -85,B 0,C 180,E1 -3342.832,E2 -3342.832} C_VEL
LIN {X 0,Y 551.737,Z 301.524,A -85,B 0,C 180,E1 -3342.974,E2 -3342.974} C_VEL
LIN {X 0,Y 551.783,Z 295.46,A -85,B 0,C 180,E1 -3345.514,E2 -3345.514} C_VEL
LIN {X 0,Y 551.839,Z 289.995,A -85,B 0,C 180,E1 -3347.797,E2 -3347.797} C_VEL
LIN {X 0,Y 551.852,Z 284.517,A -85,B 0,C 180,E1 -3350.111,E2 -3350.111} C_VEL
LIN {X 0,Y 551.885,Z 279.104,A -85,B 0,C 180,E1 -3352.459,E2 -3352.459} C_VEL
LIN {X 0,Y 551.946,Z 272.851,A -85,B 0,C 180,E1 -3355.302,E2 -3355.302} C_VEL
LIN {X 0,Y 552.037,Z 266.84,A -85,B 0,C 180,E1 -3358.102,E2 -3358.102} C_VEL
LIN {X 0,Y 552.12,Z 261.722,A -85,B 0,C 180,E1 -3360.607,E2 -3360.607} C_VEL
LIN {X 0,Y 552.245,Z 256.688,A -85,B 0,C 180,E1 -3363.176,E2 -3363.176} C_VEL
LIN {X 0,Y 552.357,Z 251.767,A -85,B 0,C 180,E1 -3365.822,E2 -3365.822} C_VEL
LIN {X 0,Y 552.446,Z 246.976,A -85,B 0,C 180,E1 -3368.561,E2 -3368.561} C_VEL
LIN {X 0,Y 552.51,Z 243.834,A -85,B 0,C 180,E1 -3370.444,E2 -3370.444} C_VEL
LIN {X 0,Y 552.511,Z 240.689,A -85,B 0,C 180,E1 -3372.456,E2 -3372.456} C_VEL
LIN {X 0,Y 552.137,Z 237.7,A -85,B 0,C 180,E1 -3374.534,E2 -3374.534} C_VEL
LIN {X 0,Y 552.086,Z 237.216,A -85,B 0,C 180,E1 -3375.559,E2 -3375.559} C_VEL
LIN {X 0,Y 552.11,Z 237.212,A -85,B 0,C 180,E1 -3378.678,E2 -3378.678} C_VEL
LIN {X 0,Y 552.115,Z 237.208,A -85,B 0,C 180,E1 -3381.408,E2 -3381.408} C_VEL
LIN {X 0,Y 552.073,Z 237.221,A -85,B 0,C 180,E1 -3384.153,E2 -3384.153} C_VEL
LIN {X 0,Y 552.115,Z 237.206,A -85,B 0,C 180,E1 -3386.811,E2 -3386.811} C_VEL
LIN {X 0,Y 552.094,Z 237.21,A -85,B 0,C 180,E1 -3389.387,E2 -3389.387} C_VEL
LIN {X 0,Y 552.077,Z 237.22,A -85,B 0,C 180,E1 -3391.897,E2 -3391.897} C_VEL
LIN {X 0,Y 552.121,Z 237.205,A -85,B 0,C 180,E1 -3394.654,E2 -3394.654} C_VEL
LIN {X 0,Y 552.088,Z 237.215,A -85,B 0,C 180,E1 -3397.546,E2 -3397.546} C_VEL
LIN {X 0,Y 552.142,Z 237.204,A -85,B 0,C 180,E1 -3400.372,E2 -3400.372} C_VEL
LIN {X 0,Y 552.118,Z 237.206,A -85,B 0,C 180,E1 -3402.973,E2 -3402.973} C_VEL
LIN {X 0,Y 552.126,Z 237.208,A -85,B 0,C 180,E1 -3406.001,E2 -3406.001} C_VEL
LIN {X 0,Y 552.153,Z 237.203,A -85,B 0,C 180,E1 -3408.99,E2 -3408.99} C_VEL
LIN {X 0,Y 552.102,Z 237.21,A -85,B 0,C 180,E1 -3411.947,E2 -3411.947} C_VEL
LIN {X 0,Y 552.175,Z 237.199,A -85,B 0,C 180,E1 -3414.152,E2 -3414.152} C_VEL
LIN {X 0,Y 552.185,Z 237.203,A -85,B 0,C 180,E1 -3417.078,E2 -3417.078} C_VEL
LIN {X 0,Y 552.208,Z 237.195,A -85,B 0,C 180,E1 -3419.996,E2 -3419.996} C_VEL
LIN {X 0,Y 552.186,Z 237.203,A -85,B 0,C 180,E1 -3422.914,E2 -3422.914} C_VEL
LIN {X 0,Y 552.17,Z 237.2,A -85,B 0,C 180,E1 -3425.84,E2 -3425.84} C_VEL
LIN {X 0,Y 552.117,Z 237.211,A -85,B 0,C 180,E1 -3428.781,E2 -3428.781} C_VEL
LIN {X 0,Y 552.143,Z 237.203,A -85,B 0,C 180,E1 -3431.746,E2 -3431.746} C_VEL
LIN {X 0,Y 552.113,Z 237.214,A -85,B 0,C 180,E1 -3434.744,E2 -3434.744} C_VEL
LIN {X 0,Y 552.073,Z 237.211,A -85,B 0,C 180,E1 -3437.784,E2 -3437.784} C_VEL
LIN {X 0,Y 552.106,Z 237.208,A -85,B 0,C 180,E1 -3440.096,E2 -3440.096} C_VEL
LIN {X 0,Y 552.062,Z 237.218,A -85,B 0,C 180,E1 -3442.446,E2 -3442.446} C_VEL
LIN {X 0,Y 552.122,Z 237.206,A -85,B 0,C 180,E1 -3445.346,E2 -3445.346} C_VEL
LIN {X 0,Y 552.091,Z 237.212,A -85,B 0,C 180,E1 -3448.093,E2 -3448.093} C_VEL
LIN {X 0,Y 552.065,Z 237.22,A -85,B 0,C 180,E1 -3450.605,E2 -3450.605} C_VEL
LIN {X 0,Y 552.089,Z 237.209,A -85,B 0,C 180,E1 -3453.18,E2 -3453.18} C_VEL
LIN {X 0,Y 552.082,Z 237.211,A -85,B 0,C 180,E1 -3453.767,E2 -3453.767} C_VEL
LIN {X 0,Y 551.446,Z 237.299,A -85,B 0,C 180,E1 -3454.376,E2 -3454.376} C_VEL
LIN {X 0,Y 548.626,Z 237.648,A -85,B 0,C 180,E1 -3455.364,E2 -3455.364} C_VEL
LIN {X 0,Y 546.204,Z 237.949,A -85,B 0,C 180,E1 -3456.16,E2 -3456.16} C_VEL
LIN {X 0,Y 545.132,Z 238.079,A -85,B 0,C 180,E1 -3456.774,E2 -3456.774} C_VEL
LIN {X 0,Y 545.027,Z 238.09,A -85,B 0,C 180,E1 -3456.982,E2 -3456.982} C_VEL
LIN {X 0,Y 545.046,Z 238.094,A -85,B 0,C 180,E1 -3460.136,E2 -3460.136} C_VEL
LIN {X 0,Y 545.022,Z 238.092,A -85,B 0,C 180,E1 -3462.694,E2 -3462.694} C_VEL
LIN {X 0,Y 545.023,Z 238.089,A -85,B 0,C 180,E1 -3465.162,E2 -3465.162} C_VEL
LIN {X 0,Y 545.038,Z 238.094,A -85,B 0,C 180,E1 -3467.894,E2 -3467.894} C_VEL
LIN {X 0,Y 545.039,Z 238.088,A -85,B 0,C 180,E1 -3470.816,E2 -3470.816} C_VEL
LIN {X 0,Y 544.999,Z 238.097,A -85,B 0,C 180,E1 -3473.617,E2 -3473.617} C_VEL
LIN {X 0,Y 545.02,Z 238.092,A -85,B 0,C 180,E1 -3476.326,E2 -3476.326} C_VEL
LIN {X 0,Y 545.013,Z 238.091,A -85,B 0,C 180,E1 -3478.95,E2 -3478.95} C_VEL
LIN {X 0,Y 545.06,Z 238.091,A -85,B 0,C 180,E1 -3481.506,E2 -3481.506} C_VEL
LIN {X 0,Y 545.068,Z 238.084,A -85,B 0,C 180,E1 -3484.48,E2 -3484.48} C_VEL
LIN {X 0,Y 545.018,Z 238.094,A -85,B 0,C 180,E1 -3487.242,E2 -3487.242} C_VEL
LIN {X 0,Y 545.054,Z 238.085,A -85,B 0,C 180,E1 -3490.413,E2 -3490.413} C_VEL
LIN {X 0,Y 545.079,Z 238.085,A -85,B 0,C 180,E1 -3492.75,E2 -3492.75} C_VEL
LIN {X 0,Y 545.033,Z 238.092,A -85,B 0,C 180,E1 -3495.819,E2 -3495.819} C_VEL
LIN {X 0,Y 545.078,Z 238.087,A -85,B 0,C 180,E1 -3498.849,E2 -3498.849} C_VEL
LIN {X 0,Y 545.073,Z 238.086,A -85,B 0,C 180,E1 -3501.846,E2 -3501.846} C_VEL
LIN {X 0,Y 545.115,Z 238.079,A -85,B 0,C 180,E1 -3504.08,E2 -3504.08} C_VEL
LIN {X 0,Y 545.118,Z 238.086,A -85,B 0,C 180,E1 -3507.044,E2 -3507.044} C_VEL
LIN {X 0,Y 545.129,Z 238.078,A -85,B 0,C 180,E1 -3510,E2 -3510} C_VEL
LIN {X 0,Y 545.118,Z 238.086,A -85,B 0,C 180,E1 -3512.956,E2 -3512.956} C_VEL
LIN {X 0,Y 545.115,Z 238.079,A -85,B 0,C 180,E1 -3515.92,E2 -3515.92} C_VEL
LIN {X 0,Y 545.073,Z 238.086,A -85,B 0,C 180,E1 -3518.154,E2 -3518.154} C_VEL
LIN {X 0,Y 545.078,Z 238.087,A -85,B 0,C 180,E1 -3521.151,E2 -3521.151} C_VEL
LIN {X 0,Y 545.033,Z 238.092,A -85,B 0,C 180,E1 -3524.181,E2 -3524.181} C_VEL
LIN {X 0,Y 545.074,Z 238.084,A -85,B 0,C 180,E1 -3527.447,E2 -3527.447} C_VEL
LIN {X 0,Y 545.037,Z 238.096,A -85,B 0,C 180,E1 -3530.374,E2 -3530.374} C_VEL
LIN {X 0,Y 545.086,Z 238.082,A -85,B 0,C 180,E1 -3533.558,E2 -3533.558} C_VEL
LIN {X 0,Y 545.043,Z 238.091,A -85,B 0,C 180,E1 -3536.002,E2 -3536.002} C_VEL
LIN {X 0,Y 545.047,Z 238.089,A -85,B 0,C 180,E1 -3538.755,E2 -3538.755} C_VEL
LIN {X 0,Y 545.018,Z 238.092,A -85,B 0,C 180,E1 -3541.686,E2 -3541.686} C_VEL
LIN {X 0,Y 545.027,Z 238.092,A -85,B 0,C 180,E1 -3544.566,E2 -3544.566} C_VEL
LIN {X 0,Y 544.987,Z 238.094,A -85,B 0,C 180,E1 -3547.307,E2 -3547.307} C_VEL
LIN {X 0,Y 545.08,Z 238.089,A -85,B 0,C 180,E1 -3550.14,E2 -3550.14} C_VEL
LIN {X 0,Y 545.035,Z 238.088,A -85,B 0,C 180,E1 -3553.11,E2 -3553.11} C_VEL
LIN {X 0,Y 545.03,Z 238.092,A -85,B 0,C 180,E1 -3556.227,E2 -3556.227} C_VEL
LIN {X 0,Y 545.076,Z 238.083,A -85,B 0,C 180,E1 -3558.894,E2 -3558.894} C_VEL
LIN {X 0,Y 545.009,Z 238.1,A -85,B 0,C 180,E1 -3561.767,E2 -3561.767} C_VEL
LIN {X 0,Y 545.023,Z 238.089,A -85,B 0,C 180,E1 -3564.538,E2 -3564.538} C_VEL
LIN {X 0,Y 545.043,Z 238.091,A -85,B 0,C 180,E1 -3567.217,E2 -3567.217} C_VEL
LIN {X 0,Y 545.026,Z 238.094,A -85,B 0,C 180,E1 -3569.815,E2 -3569.815} C_VEL
LIN {X 0,Y 545.059,Z 238.085,A -85,B 0,C 180,E1 -3572.349,E2 -3572.349} C_VEL
LIN {X 0,Y 545.084,Z 238.084,A -85,B 0,C 180,E1 -3574.825,E2 -3574.825} C_VEL
LIN {X 0,Y 545.008,Z 238.099,A -85,B 0,C 180,E1 -3577.247,E2 -3577.247} C_VEL
LIN {X 0,Y 545.093,Z 238.081,A -85,B 0,C 180,E1 -3580.42,E2 -3580.42} C_VEL
LIN {X 0,Y 545.046,Z 238.09,A -85,B 0,C 180,E1 -3583.526,E2 -3583.526} C_VEL
LIN {X 0,Y 545.069,Z 238.084,A -85,B 0,C 180,E1 -3585.825,E2 -3585.825} C_VEL
LIN {X 0,Y 545.11,Z 238.085,A -85,B 0,C 180,E1 -3588.854,E2 -3588.854} C_VEL
LIN {X 0,Y 545.076,Z 238.083,A -85,B 0,C 180,E1 -3591.851,E2 -3591.851} C_VEL
LIN {X 0,Y 545.181,Z 238.078,A -85,B 0,C 180,E1 -3594.827,E2 -3594.827} C_VEL
LIN {X 0,Y 545.17,Z 238.071,A -85,B 0,C 180,E1 -3597.788,E2 -3597.788} C_VEL
LIN {X 0,Y 545.205,Z 238.076,A -85,B 0,C 180,E1 -3600.743,E2 -3600.743} C_VEL
LIN {X 0,Y 545.15,Z 238.079,A -85,B 0,C 180,E1 -3602.96,E2 -3602.96} C_VEL
LIN {X 0,Y 545.127,Z 238.077,A -85,B 0,C 180,E1 -3605.924,E2 -3605.924} C_VEL
LIN {X 0,Y 545.06,Z 238.088,A -85,B 0,C 180,E1 -3608.158,E2 -3608.158} C_VEL
LIN {X 0,Y 545.11,Z 238.079,A -85,B 0,C 180,E1 -3611.155,E2 -3611.155} C_VEL
LIN {X 0,Y 545.088,Z 238.087,A -85,B 0,C 180,E1 -3614.184,E2 -3614.184} C_VEL
LIN {X 0,Y 545.064,Z 238.084,A -85,B 0,C 180,E1 -3617.422,E2 -3617.422} C_VEL
LIN {X 0,Y 545.089,Z 238.089,A -85,B 0,C 180,E1 -3620.376,E2 -3620.376} C_VEL
LIN {X 0,Y 545.077,Z 238.084,A -85,B 0,C 180,E1 -3623.563,E2 -3623.563} C_VEL
LIN {X 0,Y 545.056,Z 238.093,A -85,B 0,C 180,E1 -3626.005,E2 -3626.005} C_VEL
LIN {X 0,Y 545.065,Z 238.085,A -85,B 0,C 180,E1 -3628.746,E2 -3628.746} C_VEL
LIN {X 0,Y 545.06,Z 238.089,A -85,B 0,C 180,E1 -3631.681,E2 -3631.681} C_VEL
LIN {X 0,Y 545.052,Z 238.087,A -85,B 0,C 180,E1 -3634.568,E2 -3634.568} C_VEL
LIN {X 0,Y 545.032,Z 238.092,A -85,B 0,C 180,E1 -3637.307,E2 -3637.307} C_VEL
LIN {X 0,Y 545.066,Z 238.09,A -85,B 0,C 180,E1 -3640.145,E2 -3640.145} C_VEL
LIN {X 0,Y 545.043,Z 238.091,A -85,B 0,C 180,E1 -3642.696,E2 -3642.696} C_VEL
LIN {X 0,Y 545.045,Z 238.094,A -85,B 0,C 180,E1 -3644.832,E2 -3644.832} C_VEL
LIN {X 0,Y 545.48,Z 241.487,A -85,B 0,C 180,E1 -3647.258,E2 -3647.258} C_VEL
LIN {X 0,Y 545.524,Z 245.581,A -85,B 0,C 180,E1 -3649.899,E2 -3649.899} C_VEL
LIN {X 0,Y 545.404,Z 250.808,A -85,B 0,C 180,E1 -3653.03,E2 -3653.03} C_VEL
LIN {X 0,Y 545.278,Z 255.371,A -85,B 0,C 180,E1 -3655.579,E2 -3655.579} C_VEL
LIN {X 0,Y 545.161,Z 260.514,A -85,B 0,C 180,E1 -3658.306,E2 -3658.306} C_VEL
LIN {X 0,Y 545.024,Z 266.431,A -85,B 0,C 180,E1 -3661.267,E2 -3661.267} C_VEL
LIN {X 0,Y 544.921,Z 272.096,A -85,B 0,C 180,E1 -3663.992,E2 -3663.992} C_VEL
LIN {X 0,Y 544.838,Z 277.347,A -85,B 0,C 180,E1 -3666.43,E2 -3666.43} C_VEL
LIN {X 0,Y 544.809,Z 282.608,A -85,B 0,C 180,E1 -3668.827,E2 -3668.827} C_VEL
LIN {X 0,Y 544.767,Z 288.079,A -85,B 0,C 180,E1 -3671.185,E2 -3671.185} C_VEL
LIN {X 0,Y 544.704,Z 293.55,A -85,B 0,C 180,E1 -3673.51,E2 -3673.51} C_VEL
LIN {X 0,Y 544.693,Z 299.009,A -85,B 0,C 180,E1 -3675.81,E2 -3675.81} C_VEL
LIN {X 0,Y 544.638,Z 301.507,A -85,B 0,C 180,E1 -3676.854,E2 -3676.854} C_VEL
LIN {X 0,Y 546.124,Z 311.047,A -85,B 0,C 180,E1 -3677.104,E2 -3677.104} C_VEL
LIN {X 0,Y 545.994,Z 321.01,A -85,B 0,C 180,E1 -3677.408,E2 -3677.408} C_VEL
LIN {X 0,Y 545.795,Z 331.357,A -85,B 0,C 180,E1 -3677.828,E2 -3677.828} C_VEL
LIN {X 0,Y 545.598,Z 341.439,A -85,B 0,C 180,E1 -3678.351,E2 -3678.351} C_VEL
LIN {X 0,Y 545.508,Z 349.45,A -85,B 0,C 180,E1 -3678.858,E2 -3678.858} C_VEL
LIN {X 0,Y 545.372,Z 358.154,A -85,B 0,C 180,E1 -3679.513,E2 -3679.513} C_VEL
LIN {X 0,Y 545.22,Z 365.525,A -85,B 0,C 180,E1 -3680.166,E2 -3680.166} C_VEL
LIN {X 0,Y 545.101,Z 372.717,A -85,B 0,C 180,E1 -3680.913,E2 -3680.913} C_VEL
LIN {X 0,Y 544.978,Z 378.893,A -85,B 0,C 180,E1 -3681.658,E2 -3681.658} C_VEL
LIN {X 0,Y 544.84,Z 385.401,A -85,B 0,C 180,E1 -3682.589,E2 -3682.589} C_VEL
LIN {X 0,Y 544.764,Z 390.269,A -85,B 0,C 180,E1 -3683.408,E2 -3683.408} C_VEL
LIN {X 0,Y 544.739,Z 395.339,A -85,B 0,C 180,E1 -3684.447,E2 -3684.447} C_VEL
LIN {X 0,Y 544.665,Z 399.633,A -85,B 0,C 180,E1 -3685.56,E2 -3685.56} C_VEL
LIN {X 0,Y 544.67,Z 401.975,A -85,B 0,C 180,E1 -3686.301,E2 -3686.301} C_VEL
LIN {X 0,Y 544.652,Z 403.765,A -85,B 0,C 180,E1 -3687.041,E2 -3687.041} C_VEL
LIN {X 0,Y 544.546,Z 406.192,A -85,B 0,C 180,E1 -3688.521,E2 -3688.521} C_VEL
LIN {X 0,Y 544.542,Z 406.775,A -85,B 0,C 180,E1 -3689.261,E2 -3689.261} C_VEL
LIN {X 0,Y 544.542,Z 406.775,A -85,B 0,C 180,E1 -3690.739,E2 -3690.739} C_VEL
LIN {X 0,Y 544.546,Z 406.192,A -85,B 0,C 180,E1 -3691.479,E2 -3691.479} C_VEL
LIN {X 0,Y 544.652,Z 403.765,A -85,B 0,C 180,E1 -3692.959,E2 -3692.959} C_VEL
LIN {X 0,Y 544.685,Z 400.841,A -85,B 0,C 180,E1 -3694.069,E2 -3694.069} C_VEL
LIN {X 0,Y 544.654,Z 396.883,A -85,B 0,C 180,E1 -3695.182,E2 -3695.182} C_VEL
LIN {X 0,Y 544.761,Z 392.646,A -85,B 0,C 180,E1 -3696.127,E2 -3696.127} C_VEL
LIN {X 0,Y 544.826,Z 386.551,A -85,B 0,C 180,E1 -3697.225,E2 -3697.225} C_VEL
LIN {X 0,Y 544.923,Z 380.263,A -85,B 0,C 180,E1 -3698.156,E2 -3698.156} C_VEL
LIN {X 0,Y 545.041,Z 374.337,A -85,B 0,C 180,E1 -3698.901,E2 -3698.901} C_VEL
LIN {X 0,Y 545.201,Z 367.438,A -85,B 0,C 180,E1 -3699.647,E2 -3699.647} C_VEL
LIN {X 0,Y 545.344,Z 359.286,A -85,B 0,C 180,E1 -3700.394,E2 -3700.394} C_VEL
LIN {X 0,Y 545.483,Z 350.799,A -85,B 0,C 180,E1 -3701.049,E2 -3701.049} C_VEL
LIN {X 0,Y 545.596,Z 341.499,A -85,B 0,C 180,E1 -3701.646,E2 -3701.646} C_VEL
LIN {X 0,Y 545.826,Z 331.357,A -85,B 0,C 180,E1 -3702.171,E2 -3702.171} C_VEL
LIN {X 0,Y 545.99,Z 322.296,A -85,B 0,C 180,E1 -3702.545,E2 -3702.545} C_VEL
LIN {X 0,Y 546.125,Z 312.795,A -85,B 0,C 180,E1 -3702.849,E2 -3702.849} C_VEL
LIN {X 0,Y 545.77,Z 307.987,A -85,B 0,C 180,E1 -3702.988,E2 -3702.988} C_VEL
LIN {X 0,Y 544.638,Z 301.507,A -85,B 0,C 180,E1 -3703.146,E2 -3703.146} C_VEL
LIN {X 0,Y 544.686,Z 295.371,A -85,B 0,C 180,E1 -3705.721,E2 -3705.721} C_VEL
LIN {X 0,Y 544.748,Z 289.904,A -85,B 0,C 180,E1 -3708.037,E2 -3708.037} C_VEL
LIN {X 0,Y 544.793,Z 284.426,A -85,B 0,C 180,E1 -3710.383,E2 -3710.383} C_VEL
LIN {X 0,Y 544.828,Z 279.101,A -85,B 0,C 180,E1 -3712.766,E2 -3712.766} C_VEL
LIN {X 0,Y 544.887,Z 273.244,A -85,B 0,C 180,E1 -3715.46,E2 -3715.46} C_VEL
LIN {X 0,Y 544.972,Z 268.596,A -85,B 0,C 180,E1 -3717.662,E2 -3717.662} C_VEL
LIN {X 0,Y 545.105,Z 263.338,A -85,B 0,C 180,E1 -3720.249,E2 -3720.249} C_VEL
LIN {X 0,Y 545.235,Z 257.838,A -85,B 0,C 180,E1 -3723.085,E2 -3723.085} C_VEL
LIN {X 0,Y 545.338,Z 253.007,A -85,B 0,C 180,E1 -3725.715,E2 -3725.715} C_VEL
LIN {X 0,Y 545.419,Z 248.689,A -85,B 0,C 180,E1 -3728.206,E2 -3728.206} C_VEL
LIN {X 0,Y 545.501,Z 244.877,A -85,B 0,C 180,E1 -3730.522,E2 -3730.522} C_VEL
LIN {X 0,Y 545.442,Z 241.007,A -85,B 0,C 180,E1 -3733.07,E2 -3733.07} C_VEL
LIN {X 0,Y 545.043,Z 238.094,A -85,B 0,C 180,E1 -3735.168,E2 -3735.168} C_VEL
LIN {X 0,Y 545.072,Z 238.092,A -85,B 0,C 180,E1 -3738.402,E2 -3738.402} C_VEL
LIN {X 0,Y 545.079,Z 238.086,A -85,B 0,C 180,E1 -3740.815,E2 -3740.815} C_VEL
LIN {X 0,Y 545.035,Z 238.092,A -85,B 0,C 180,E1 -3743.616,E2 -3743.616} C_VEL
LIN {X 0,Y 545.065,Z 238.089,A -85,B 0,C 180,E1 -3746.325,E2 -3746.325} C_VEL
LIN {X 0,Y 545.064,Z 238.084,A -85,B 0,C 180,E1 -3748.949,E2 -3748.949} C_VEL
LIN {X 0,Y 545.055,Z 238.088,A -85,B 0,C 180,E1 -3751.502,E2 -3751.502} C_VEL
LIN {X 0,Y 545.093,Z 238.081,A -85,B 0,C 180,E1 -3754.816,E2 -3754.816} C_VEL
LIN {X 0,Y 545.033,Z 238.09,A -85,B 0,C 180,E1 -3757.239,E2 -3757.239} C_VEL
LIN {X 0,Y 545.114,Z 238.079,A -85,B 0,C 180,E1 -3760.411,E2 -3760.411} C_VEL
LIN {X 0,Y 545.05,Z 238.093,A -85,B 0,C 180,E1 -3763.517,E2 -3763.517} C_VEL
LIN {X 0,Y 545.088,Z 238.087,A -85,B 0,C 180,E1 -3765.816,E2 -3765.816} C_VEL
LIN {X 0,Y 545.11,Z 238.079,A -85,B 0,C 180,E1 -3768.845,E2 -3768.845} C_VEL
LIN {X 0,Y 545.06,Z 238.088,A -85,B 0,C 180,E1 -3771.842,E2 -3771.842} C_VEL
LIN {X 0,Y 545.127,Z 238.077,A -85,B 0,C 180,E1 -3774.076,E2 -3774.076} C_VEL
LIN {X 0,Y 545.15,Z 238.079,A -85,B 0,C 180,E1 -3777.04,E2 -3777.04} C_VEL
LIN {X 0,Y 545.18,Z 238.07,A -85,B 0,C 180,E1 -3779.996,E2 -3779.996} C_VEL
LIN {X 0,Y 545.153,Z 238.079,A -85,B 0,C 180,E1 -3782.951,E2 -3782.951} C_VEL
LIN {X 0,Y 545.119,Z 238.078,A -85,B 0,C 180,E1 -3785.915,E2 -3785.915} C_VEL
LIN {X 0,Y 545.076,Z 238.083,A -85,B 0,C 180,E1 -3788.149,E2 -3788.149} C_VEL
LIN {X 0,Y 545.124,Z 238.078,A -85,B 0,C 180,E1 -3791.535,E2 -3791.535} C_VEL
LIN {X 0,Y 545.079,Z 238.09,A -85,B 0,C 180,E1 -3794.762,E2 -3794.762} C_VEL
LIN {X 0,Y 545.049,Z 238.087,A -85,B 0,C 180,E1 -3797.417,E2 -3797.417} C_VEL
LIN {X 0,Y 545.07,Z 238.087,A -85,B 0,C 180,E1 -3800.367,E2 -3800.367} C_VEL
LIN {X 0,Y 545.049,Z 238.086,A -85,B 0,C 180,E1 -3803.555,E2 -3803.555} C_VEL
LIN {X 0,Y 545.045,Z 238.088,A -85,B 0,C 180,E1 -3805.996,E2 -3805.996} C_VEL
LIN {X 0,Y 545.056,Z 238.091,A -85,B 0,C 180,E1 -3808.744,E2 -3808.744} C_VEL
LIN {X 0,Y 545.02,Z 238.09,A -85,B 0,C 180,E1 -3811.674,E2 -3811.674} C_VEL
LIN {X 0,Y 545.043,Z 238.093,A -85,B 0,C 180,E1 -3814.558,E2 -3814.558} C_VEL
LIN {X 0,Y 545.027,Z 238.09,A -85,B 0,C 180,E1 -3816.982,E2 -3816.982} C_VEL
LIN {X 0,Y 544.317,Z 238.179,A -85,B 0,C 180,E1 -3817.598,E2 -3817.598} C_VEL
LIN {X 0,Y 541.461,Z 238.537,A -85,B 0,C 180,E1 -3818.599,E2 -3818.599} C_VEL
LIN {X 0,Y 539.083,Z 238.832,A -85,B 0,C 180,E1 -3819.405,E2 -3819.405} C_VEL
LIN {X 0,Y 538.077,Z 238.961,A -85,B 0,C 180,E1 -3820.027,E2 -3820.027} C_VEL
LIN {X 0,Y 538.001,Z 238.964,A -85,B 0,C 180,E1 -3820.238,E2 -3820.238} C_VEL
LIN {X 0,Y 538.017,Z 238.962,A -85,B 0,C 180,E1 -3822.988,E2 -3822.988} C_VEL
LIN {X 0,Y 537.981,Z 238.973,A -85,B 0,C 180,E1 -3825.921,E2 -3825.921} C_VEL
LIN {X 0,Y 538.027,Z 238.961,A -85,B 0,C 180,E1 -3829.245,E2 -3829.245} C_VEL
LIN {X 0,Y 537.941,Z 238.978,A -85,B 0,C 180,E1 -3832.119,E2 -3832.119} C_VEL
LIN {X 0,Y 537.964,Z 238.969,A -85,B 0,C 180,E1 -3834.914,E2 -3834.914} C_VEL
LIN {X 0,Y 537.973,Z 238.974,A -85,B 0,C 180,E1 -3837.615,E2 -3837.615} C_VEL
LIN {X 0,Y 537.988,Z 238.968,A -85,B 0,C 180,E1 -3840.238,E2 -3840.238} C_VEL
LIN {X 0,Y 538.009,Z 238.963,A -85,B 0,C 180,E1 -3842.794,E2 -3842.794} C_VEL
LIN {X 0,Y 538.009,Z 238.967,A -85,B 0,C 180,E1 -3845.291,E2 -3845.291} C_VEL
LIN {X 0,Y 537.982,Z 238.969,A -85,B 0,C 180,E1 -3848.031,E2 -3848.031} C_VEL
LIN {X 0,Y 537.979,Z 238.969,A -85,B 0,C 180,E1 -3850.938,E2 -3850.938} C_VEL
LIN {X 0,Y 537.995,Z 238.974,A -85,B 0,C 180,E1 -3853.298,E2 -3853.298} C_VEL
LIN {X 0,Y 537.999,Z 238.971,A -85,B 0,C 180,E1 -3855.629,E2 -3855.629} C_VEL
LIN {X 0,Y 538.031,Z 238.963,A -85,B 0,C 180,E1 -3858.701,E2 -3858.701} C_VEL
LIN {X 0,Y 538.029,Z 238.964,A -85,B 0,C 180,E1 -3861.739,E2 -3861.739} C_VEL
LIN {X 0,Y 538.067,Z 238.958,A -85,B 0,C 180,E1 -3864.002,E2 -3864.002} C_VEL
LIN {X 0,Y 538.083,Z 238.962,A -85,B 0,C 180,E1 -3867.005,E2 -3867.005} C_VEL
LIN {X 0,Y 538.099,Z 238.954,A -85,B 0,C 180,E1 -3870,E2 -3870} C_VEL
LIN {X 0,Y 538.083,Z 238.962,A -85,B 0,C 180,E1 -3872.995,E2 -3872.995} C_VEL
LIN {X 0,Y 538.067,Z 238.958,A -85,B 0,C 180,E1 -3875.998,E2 -3875.998} C_VEL
LIN {X 0,Y 538.029,Z 238.964,A -85,B 0,C 180,E1 -3878.261,E2 -3878.261} C_VEL
LIN {X 0,Y 538.031,Z 238.961,A -85,B 0,C 180,E1 -3881.608,E2 -3881.608} C_VEL
LIN {X 0,Y 538.015,Z 238.969,A -85,B 0,C 180,E1 -3884.869,E2 -3884.869} C_VEL
LIN {X 0,Y 538.025,Z 238.962,A -85,B 0,C 180,E1 -3887.554,E2 -3887.554} C_VEL
LIN {X 0,Y 537.979,Z 238.973,A -85,B 0,C 180,E1 -3890.653,E2 -3890.653} C_VEL
LIN {X 0,Y 538.013,Z 238.965,A -85,B 0,C 180,E1 -3893.887,E2 -3893.887} C_VEL
LIN {X 0,Y 537.996,Z 238.974,A -85,B 0,C 180,E1 -3896.368,E2 -3896.368} C_VEL
LIN {X 0,Y 538.013,Z 238.964,A -85,B 0,C 180,E1 -3898.945,E2 -3898.945} C_VEL
LIN {X 0,Y 537.969,Z 238.973,A -85,B 0,C 180,E1 -3901.894,E2 -3901.894} C_VEL
LIN {X 0,Y 537.977,Z 238.97,A -85,B 0,C 180,E1 -3904.625,E2 -3904.625} C_VEL
LIN {X 0,Y 537.953,Z 238.97,A -85,B 0,C 180,E1 -3907.175,E2 -3907.175} C_VEL
LIN {X 0,Y 538.041,Z 238.965,A -85,B 0,C 180,E1 -3909.794,E2 -3909.794} C_VEL
LIN {X 0,Y 537.971,Z 238.968,A -85,B 0,C 180,E1 -3912.789,E2 -3912.789} C_VEL
LIN {X 0,Y 537.994,Z 238.973,A -85,B 0,C 180,E1 -3915.928,E2 -3915.928} C_VEL
LIN {X 0,Y 538.012,Z 238.966,A -85,B 0,C 180,E1 -3918.234,E2 -3918.234} C_VEL
LIN {X 0,Y 537.97,Z 238.97,A -85,B 0,C 180,E1 -3921.174,E2 -3921.174} C_VEL
LIN {X 0,Y 537.988,Z 238.969,A -85,B 0,C 180,E1 -3924.088,E2 -3924.088} C_VEL
LIN {X 0,Y 537.996,Z 238.965,A -85,B 0,C 180,E1 -3926.733,E2 -3926.733} C_VEL
LIN {X 0,Y 537.988,Z 238.975,A -85,B 0,C 180,E1 -3929.561,E2 -3929.561} C_VEL
LIN {X 0,Y 538.012,Z 238.965,A -85,B 0,C 180,E1 -3931.955,E2 -3931.955} C_VEL
LIN {X 0,Y 538.037,Z 238.96,A -85,B 0,C 180,E1 -3934.472,E2 -3934.472} C_VEL
LIN {X 0,Y 537.963,Z 238.972,A -85,B 0,C 180,E1 -3937.743,E2 -3937.743} C_VEL
LIN {X 0,Y 538.052,Z 238.958,A -85,B 0,C 180,E1 -3940.153,E2 -3940.153} C_VEL
LIN {X 0,Y 537.993,Z 238.972,A -85,B 0,C 180,E1 -3943.304,E2 -3943.304} C_VEL
LIN {X 0,Y 538.039,Z 238.962,A -85,B 0,C 180,E1 -3945.635,E2 -3945.635} C_VEL
LIN {X 0,Y 538.068,Z 238.96,A -85,B 0,C 180,E1 -3948.707,E2 -3948.707} C_VEL
LIN {X 0,Y 538.04,Z 238.96,A -85,B 0,C 180,E1 -3951.744,E2 -3951.744} C_VEL
LIN {X 0,Y 538.136,Z 238.954,A -85,B 0,C 180,E1 -3954.759,E2 -3954.759} C_VEL
LIN {X 0,Y 538.143,Z 238.946,A -85,B 0,C 180,E1 -3957.759,E2 -3957.759} C_VEL
LIN {X 0,Y 538.174,Z 238.952,A -85,B 0,C 180,E1 -3960.753,E2 -3960.753} C_VEL
LIN {X 0,Y 538.116,Z 238.954,A -85,B 0,C 180,E1 -3962.999,E2 -3962.999} C_VEL
LIN {X 0,Y 538.083,Z 238.955,A -85,B 0,C 180,E1 -3966.002,E2 -3966.002} C_VEL
LIN {X 0,Y 538.032,Z 238.965,A -85,B 0,C 180,E1 -3968.265,E2 -3968.265} C_VEL
LIN {X 0,Y 538.08,Z 238.954,A -85,B 0,C 180,E1 -3971.602,E2 -3971.602} C_VEL
LIN {X 0,Y 538.056,Z 238.96,A -85,B 0,C 180,E1 -3974.861,E2 -3974.861} C_VEL
LIN {X 0,Y 538.034,Z 238.96,A -85,B 0,C 180,E1 -3977.536,E2 -3977.536} C_VEL
LIN {X 0,Y 538.034,Z 238.963,A -85,B 0,C 180,E1 -3980.655,E2 -3980.655} C_VEL
LIN {X 0,Y 538.008,Z 238.968,A -85,B 0,C 180,E1 -3983.881,E2 -3983.881} C_VEL
LIN {X 0,Y 538.01,Z 238.968,A -85,B 0,C 180,E1 -3986.371,E2 -3986.371} C_VEL
LIN {X 0,Y 538.032,Z 238.96,A -85,B 0,C 180,E1 -3988.936,E2 -3988.936} C_VEL
LIN {X 0,Y 538.012,Z 238.971,A -85,B 0,C 180,E1 -3991.89,E2 -3991.89} C_VEL
LIN {X 0,Y 538.002,Z 238.965,A -85,B 0,C 180,E1 -3994.618,E2 -3994.618} C_VEL
LIN {X 0,Y 538.001,Z 238.967,A -85,B 0,C 180,E1 -3997.171,E2 -3997.171} C_VEL
LIN {X 0,Y 538.012,Z 238.972,A -85,B 0,C 180,E1 -3999.801,E2 -3999.801} C_VEL
LIN {X 0,Y 537.993,Z 238.97,A -85,B 0,C 180,E1 -4002.791,E2 -4002.791} C_VEL
LIN {X 0,Y 538.018,Z 238.97,A -85,B 0,C 180,E1 -4004.075,E2 -4004.075} C_VEL
LIN {X 0,Y 538.111,Z 239.74,A -85,B 0,C 180,E1 -4005.15,E2 -4005.15} C_VEL
LIN {X 0,Y 538.482,Z 242.69,A -85,B 0,C 180,E1 -4007.261,E2 -4007.261} C_VEL
LIN {X 0,Y 538.517,Z 245.729,A -85,B 0,C 180,E1 -4009.268,E2 -4009.268} C_VEL
LIN {X 0,Y 538.388,Z 250.419,A -85,B 0,C 180,E1 -4012.156,E2 -4012.156} C_VEL
LIN {X 0,Y 538.289,Z 255.227,A -85,B 0,C 180,E1 -4014.938,E2 -4014.938} C_VEL
LIN {X 0,Y 538.161,Z 260.163,A -85,B 0,C 180,E1 -4017.628,E2 -4017.628} C_VEL
LIN {X 0,Y 538.024,Z 265.212,A -85,B 0,C 180,E1 -4020.24,E2 -4020.24} C_VEL
LIN {X 0,Y 537.922,Z 270.351,A -85,B 0,C 180,E1 -4022.789,E2 -4022.789} C_VEL
LIN {X 0,Y 537.813,Z 275.564,A -85,B 0,C 180,E1 -4025.282,E2 -4025.282} C_VEL
LIN {X 0,Y 537.755,Z 282.605,A -85,B 0,C 180,E1 -4028.535,E2 -4028.535} C_VEL
LIN {X 0,Y 537.694,Z 287.988,A -85,B 0,C 180,E1 -4030.928,E2 -4030.928} C_VEL
LIN {X 0,Y 537.639,Z 293.46,A -85,B 0,C 180,E1 -4033.287,E2 -4033.287} C_VEL
LIN {X 0,Y 537.563,Z 300.738,A -85,B 0,C 180,E1 -4036.389,E2 -4036.389} C_VEL
LIN {X 0,Y 537.57,Z 301.589,A -85,B 0,C 180,E1 -4036.69,E2 -4036.69} C_VEL
LIN {X 0,Y 539.204,Z 311.74,A -85,B 0,C 180,E1 -4036.959,E2 -4036.959} C_VEL
LIN {X 0,Y 539.047,Z 320.842,A -85,B 0,C 180,E1 -4037.243,E2 -4037.243} C_VEL
LIN {X 0,Y 538.862,Z 331.207,A -85,B 0,C 180,E1 -4037.669,E2 -4037.669} C_VEL
LIN {X 0,Y 538.63,Z 341.384,A -85,B 0,C 180,E1 -4038.202,E2 -4038.202} C_VEL
LIN {X 0,Y 538.491,Z 350.697,A -85,B 0,C 180,E1 -4038.806,E2 -4038.806} C_VEL
LIN {X 0,Y 538.344,Z 359.212,A -85,B 0,C 180,E1 -4039.469,E2 -4039.469} C_VEL
LIN {X 0,Y 538.129,Z 367.393,A -85,B 0,C 180,E1 -4040.225,E2 -4040.225} C_VEL
LIN {X 0,Y 537.966,Z 375.948,A -85,B 0,C 180,E1 -4041.17,E2 -4041.17} C_VEL
LIN {X 0,Y 537.82,Z 384.243,A -85,B 0,C 180,E1 -4042.303,E2 -4042.303} C_VEL
LIN {X 0,Y 537.701,Z 390.648,A -85,B 0,C 180,E1 -4043.398,E2 -4043.398} C_VEL
LIN {X 0,Y 537.674,Z 395.331,A -85,B 0,C 180,E1 -4044.374,E2 -4044.374} C_VEL
LIN {X 0,Y 537.563,Z 399.626,A -85,B 0,C 180,E1 -4045.501,E2 -4045.501} C_VEL
LIN {X 0,Y 537.592,Z 401.973,A -85,B 0,C 180,E1 -4046.252,E2 -4046.252} C_VEL
LIN {X 0,Y 537.552,Z 403.759,A -85,B 0,C 180,E1 -4047.002,E2 -4047.002} C_VEL
LIN {X 0,Y 537.452,Z 406.184,A -85,B 0,C 180,E1 -4048.501,E2 -4048.501} C_VEL
LIN {X 0,Y 537.442,Z 406.768,A -85,B 0,C 180,E1 -4049.251,E2 -4049.251} C_VEL
LIN {X 0,Y 537.442,Z 406.768,A -85,B 0,C 180,E1 -4050.749,E2 -4050.749} C_VEL
LIN {X 0,Y 537.452,Z 406.184,A -85,B 0,C 180,E1 -4051.499,E2 -4051.499} C_VEL
LIN {X 0,Y 537.552,Z 403.759,A -85,B 0,C 180,E1 -4052.998,E2 -4052.998} C_VEL
LIN {X 0,Y 537.606,Z 400.834,A -85,B 0,C 180,E1 -4054.123,E2 -4054.123} C_VEL
LIN {X 0,Y 537.588,Z 396.875,A -85,B 0,C 180,E1 -4055.25,E2 -4055.25} C_VEL
LIN {X 0,Y 537.64,Z 392.096,A -85,B 0,C 180,E1 -4056.316,E2 -4056.316} C_VEL
LIN {X 0,Y 537.758,Z 386.542,A -85,B 0,C 180,E1 -4057.321,E2 -4057.321} C_VEL
LIN {X 0,Y 537.885,Z 380.255,A -85,B 0,C 180,E1 -4058.263,E2 -4058.263} C_VEL
LIN {X 0,Y 537.999,Z 374.322,A -85,B 0,C 180,E1 -4059.019,E2 -4059.019} C_VEL
LIN {X 0,Y 538.16,Z 367.394,A -85,B 0,C 180,E1 -4059.774,E2 -4059.774} C_VEL
LIN {X 0,Y 538.344,Z 359.212,A -85,B 0,C 180,E1 -4060.531,E2 -4060.531} C_VEL
LIN {X 0,Y 538.501,Z 350.697,A -85,B 0,C 180,E1 -4061.194,E2 -4061.194} C_VEL
LIN {X 0,Y 538.601,Z 342.328,A -85,B 0,C 180,E1 -4061.743,E2 -4061.743} C_VEL
LIN {X 0,Y 538.84,Z 332.214,A -85,B 0,C 180,E1 -4062.284,E2 -4062.284} C_VEL
LIN {X 0,Y 539.019,Z 323.418,A -85,B 0,C 180,E1 -4062.662,E2 -4062.662} C_VEL
LIN {X 0,Y 539.177,Z 313.489,A -85,B 0,C 180,E1 -4062.994,E2 -4062.994} C_VEL
LIN {X 0,Y 538.772,Z 308.666,A -85,B 0,C 180,E1 -4063.135,E2 -4063.135} C_VEL
LIN {X 0,Y 537.583,Z 301.414,A -85,B 0,C 180,E1 -4063.321,E2 -4063.321} C_VEL
LIN {X 0,Y 537.62,Z 295.281,A -85,B 0,C 180,E1 -4065.933,E2 -4065.933} C_VEL
LIN {X 0,Y 537.674,Z 289.813,A -85,B 0,C 180,E1 -4068.282,E2 -4068.282} C_VEL
LIN {X 0,Y 537.71,Z 284.359,A -85,B 0,C 180,E1 -4070.664,E2 -4070.664} C_VEL
LIN {X 0,Y 537.75,Z 279.074,A -85,B 0,C 180,E1 -4073.083,E2 -4073.083} C_VEL
LIN {X 0,Y 537.844,Z 273.628,A -85,B 0,C 180,E1 -4075.625,E2 -4075.625} C_VEL
LIN {X 0,Y 537.934,Z 268.601,A -85,B 0,C 180,E1 -4078.055,E2 -4078.055} C_VEL
LIN {X 0,Y 538.054,Z 263.512,A -85,B 0,C 180,E1 -4080.624,E2 -4080.624} C_VEL
LIN {X 0,Y 538.221,Z 258.392,A -85,B 0,C 180,E1 -4083.309,E2 -4083.309} C_VEL
LIN {X 0,Y 538.316,Z 253.599,A -85,B 0,C 180,E1 -4085.979,E2 -4085.979} C_VEL
LIN {X 0,Y 538.424,Z 248.809,A -85,B 0,C 180,E1 -4088.794,E2 -4088.794} C_VEL
LIN {X 0,Y 538.534,Z 244.192,A -85,B 0,C 180,E1 -4091.724,E2 -4091.724} C_VEL
LIN {X 0,Y 538.265,Z 240.772,A -85,B 0,C 180,E1 -4094.098,E2 -4094.098} C_VEL
LIN {X 0,Y 538.051,Z 239.342,A -85,B 0,C 180,E1 -4095.14,E2 -4095.14} C_VEL
LIN {X 0,Y 538.005,Z 238.972,A -85,B 0,C 180,E1 -4096.181,E2 -4096.181} C_VEL
LIN {X 0,Y 538.026,Z 238.964,A -85,B 0,C 180,E1 -4099.254,E2 -4099.254} C_VEL
LIN {X 0,Y 537.99,Z 238.975,A -85,B 0,C 180,E1 -4102.119,E2 -4102.119} C_VEL
LIN {X 0,Y 537.991,Z 238.968,A -85,B 0,C 180,E1 -4104.912,E2 -4104.912} C_VEL
LIN {X 0,Y 538.019,Z 238.965,A -85,B 0,C 180,E1 -4107.614,E2 -4107.614} C_VEL
LIN {X 0,Y 538.008,Z 238.968,A -85,B 0,C 180,E1 -4110.235,E2 -4110.235} C_VEL
LIN {X 0,Y 538.004,Z 238.964,A -85,B 0,C 180,E1 -4112.79,E2 -4112.79} C_VEL
LIN {X 0,Y 538.015,Z 238.964,A -85,B 0,C 180,E1 -4115.288,E2 -4115.288} C_VEL
LIN {X 0,Y 538.015,Z 238.968,A -85,B 0,C 180,E1 -4118.039,E2 -4118.039} C_VEL
LIN {X 0,Y 538.079,Z 238.958,A -85,B 0,C 180,E1 -4120.145,E2 -4120.145} C_VEL
LIN {X 0,Y 537.998,Z 238.968,A -85,B 0,C 180,E1 -4123.295,E2 -4123.295} C_VEL
LIN {X 0,Y 538.058,Z 238.966,A -85,B 0,C 180,E1 -4125.627,E2 -4125.627} C_VEL
LIN {X 0,Y 538.07,Z 238.956,A -85,B 0,C 180,E1 -4128.698,E2 -4128.698} C_VEL
LIN {X 0,Y 538.032,Z 238.965,A -85,B 0,C 180,E1 -4131.735,E2 -4131.735} C_VEL
LIN {X 0,Y 538.083,Z 238.955,A -85,B 0,C 180,E1 -4133.998,E2 -4133.998} C_VEL
LIN {X 0,Y 538.116,Z 238.954,A -85,B 0,C 180,E1 -4137.001,E2 -4137.001} C_VEL
LIN {X 0,Y 538.151,Z 238.946,A -85,B 0,C 180,E1 -4139.996,E2 -4139.996} C_VEL
LIN {X 0,Y 538.12,Z 238.956,A -85,B 0,C 180,E1 -4142.99,E2 -4142.99} C_VEL
LIN {X 0,Y 538.074,Z 238.955,A -85,B 0,C 180,E1 -4145.993,E2 -4145.993} C_VEL
LIN {X 0,Y 538.032,Z 238.97,A -85,B 0,C 180,E1 -4149.013,E2 -4149.013} C_VEL
LIN {X 0,Y 538.062,Z 238.957,A -85,B 0,C 180,E1 -4152.058,E2 -4152.058} C_VEL
LIN {X 0,Y 538.021,Z 238.967,A -85,B 0,C 180,E1 -4155.139,E2 -4155.139} C_VEL
LIN {X 0,Y 538.001,Z 238.966,A -85,B 0,C 180,E1 -4158.265,E2 -4158.265} C_VEL
LIN {X 0,Y 538.014,Z 238.971,A -85,B 0,C 180,E1 -4160.646,E2 -4160.646} C_VEL
LIN {X 0,Y 537.972,Z 238.968,A -85,B 0,C 180,E1 -4163.884,E2 -4163.884} C_VEL
LIN {X 0,Y 538.008,Z 238.969,A -85,B 0,C 180,E1 -4166.362,E2 -4166.362} C_VEL
LIN {X 0,Y 537.996,Z 238.968,A -85,B 0,C 180,E1 -4168.929,E2 -4168.929} C_VEL
LIN {X 0,Y 537.975,Z 238.969,A -85,B 0,C 180,E1 -4171.883,E2 -4171.883} C_VEL
LIN {X 0,Y 537.993,Z 238.971,A -85,B 0,C 180,E1 -4174.617,E2 -4174.617} C_VEL
LIN {X 0,Y 537.966,Z 238.969,A -85,B 0,C 180,E1 -4177.166,E2 -4177.166} C_VEL
LIN {X 0,Y 538.001,Z 238.964,A -85,B 0,C 180,E1 -4180.238,E2 -4180.238} C_VEL
LIN {X 0,Y 537.355,Z 239.047,A -85,B 0,C 180,E1 -4180.863,E2 -4180.863} C_VEL
LIN {X 0,Y 534.518,Z 239.402,A -85,B 0,C 180,E1 -4181.877,E2 -4181.877} C_VEL
LIN {X 0,Y 532.098,Z 239.703,A -85,B 0,C 180,E1 -4182.695,E2 -4182.695} C_VEL
LIN {X 0,Y 531.042,Z 239.832,A -85,B 0,C 180,E1 -4183.325,E2 -4183.325} C_VEL
LIN {X 0,Y 530.948,Z 239.844,A -85,B 0,C 180,E1 -4183.539,E2 -4183.539} C_VEL
LIN {X 0,Y 530.915,Z 239.85,A -85,B 0,C 180,E1 -4186.502,E2 -4186.502} C_VEL
LIN {X 0,Y 530.98,Z 239.842,A -85,B 0,C 180,E1 -4189.568,E2 -4189.568} C_VEL
LIN {X 0,Y 530.913,Z 239.848,A -85,B 0,C 180,E1 -4192.573,E2 -4192.573} C_VEL
LIN {X 0,Y 530.946,Z 239.845,A -85,B 0,C 180,E1 -4195.308,E2 -4195.308} C_VEL
LIN {X 0,Y 530.924,Z 239.851,A -85,B 0,C 180,E1 -4198.03,E2 -4198.03} C_VEL
LIN {X 0,Y 530.957,Z 239.842,A -85,B 0,C 180,E1 -4200.865,E2 -4200.865} C_VEL
LIN {X 0,Y 530.953,Z 239.845,A -85,B 0,C 180,E1 -4203.254,E2 -4203.254} C_VEL
LIN {X 0,Y 530.964,Z 239.845,A -85,B 0,C 180,E1 -4205.947,E2 -4205.947} C_VEL
LIN {X 0,Y 530.943,Z 239.846,A -85,B 0,C 180,E1 -4209.06,E2 -4209.06} C_VEL
LIN {X 0,Y 530.983,Z 239.84,A -85,B 0,C 180,E1 -4212.334,E2 -4212.334} C_VEL
LIN {X 0,Y 530.984,Z 239.847,A -85,B 0,C 180,E1 -4215.435,E2 -4215.435} C_VEL
LIN {X 0,Y 530.984,Z 239.84,A -85,B 0,C 180,E1 -4218.549,E2 -4218.549} C_VEL
LIN {X 0,Y 530.998,Z 239.842,A -85,B 0,C 180,E1 -4221.629,E2 -4221.629} C_VEL
LIN {X 0,Y 531.025,Z 239.835,A -85,B 0,C 180,E1 -4223.922,E2 -4223.922} C_VEL
LIN {X 0,Y 531.049,Z 239.838,A -85,B 0,C 180,E1 -4226.966,E2 -4226.966} C_VEL
LIN {X 0,Y 531.07,Z 239.83,A -85,B 0,C 180,E1 -4230,E2 -4230} C_VEL
LIN {X 0,Y 531.049,Z 239.838,A -85,B 0,C 180,E1 -4233.034,E2 -4233.034} C_VEL
LIN {X 0,Y 531.025,Z 239.835,A -85,B 0,C 180,E1 -4236.078,E2 -4236.078} C_VEL
LIN {X 0,Y 530.998,Z 239.842,A -85,B 0,C 180,E1 -4238.371,E2 -4238.371} C_VEL
LIN {X 0,Y 530.993,Z 239.838,A -85,B 0,C 180,E1 -4241.68,E2 -4241.68} C_VEL
LIN {X 0,Y 530.98,Z 239.845,A -85,B 0,C 180,E1 -4244.965,E2 -4244.965} C_VEL
LIN {X 0,Y 530.962,Z 239.843,A -85,B 0,C 180,E1 -4247.724,E2 -4247.724} C_VEL
LIN {X 0,Y 530.943,Z 239.846,A -85,B 0,C 180,E1 -4250.94,E2 -4250.94} C_VEL
LIN {X 0,Y 530.964,Z 239.845,A -85,B 0,C 180,E1 -4254.053,E2 -4254.053} C_VEL
LIN {X 0,Y 530.953,Z 239.845,A -85,B 0,C 180,E1 -4256.746,E2 -4256.746} C_VEL
LIN {X 0,Y 530.948,Z 239.843,A -85,B 0,C 180,E1 -4259.324,E2 -4259.324} C_VEL
LIN {X 0,Y 530.922,Z 239.854,A -85,B 0,C 180,E1 -4262.107,E2 -4262.107} C_VEL
LIN {X 0,Y 530.933,Z 239.845,A -85,B 0,C 180,E1 -4264.858,E2 -4264.858} C_VEL
LIN {X 0,Y 530.913,Z 239.849,A -85,B 0,C 180,E1 -4267.511,E2 -4267.511} C_VEL
LIN {X 0,Y 530.986,Z 239.841,A -85,B 0,C 180,E1 -4270.431,E2 -4270.431} C_VEL
LIN {X 0,Y 530.915,Z 239.85,A -85,B 0,C 180,E1 -4273.498,E2 -4273.498} C_VEL
LIN {X 0,Y 530.951,Z 239.843,A -85,B 0,C 180,E1 -4276.513,E2 -4276.513} C_VEL
LIN {X 0,Y 530.981,Z 239.845,A -85,B 0,C 180,E1 -4279.576,E2 -4279.576} C_VEL
LIN {X 0,Y 530.926,Z 239.845,A -85,B 0,C 180,E1 -4282.581,E2 -4282.581} C_VEL
LIN {X 0,Y 530.962,Z 239.845,A -85,B 0,C 180,E1 -4285.316,E2 -4285.316} C_VEL
LIN {X 0,Y 530.933,Z 239.847,A -85,B 0,C 180,E1 -4288.037,E2 -4288.037} C_VEL
LIN {X 0,Y 530.953,Z 239.843,A -85,B 0,C 180,E1 -4290.879,E2 -4290.879} C_VEL
LIN {X 0,Y 530.971,Z 239.846,A -85,B 0,C 180,E1 -4293.261,E2 -4293.261} C_VEL
LIN {X 0,Y 530.953,Z 239.844,A -85,B 0,C 180,E1 -4295.966,E2 -4295.966} C_VEL
LIN {X 0,Y 530.973,Z 239.845,A -85,B 0,C 180,E1 -4299.067,E2 -4299.067} C_VEL
LIN {X 0,Y 530.961,Z 239.846,A -85,B 0,C 180,E1 -4301.484,E2 -4301.484} C_VEL
LIN {X 0,Y 530.971,Z 239.842,A -85,B 0,C 180,E1 -4304.655,E2 -4304.655} C_VEL
LIN {X 0,Y 531.019,Z 239.835,A -85,B 0,C 180,E1 -4307.78,E2 -4307.78} C_VEL
LIN {X 0,Y 530.962,Z 239.841,A -85,B 0,C 180,E1 -4310.097,E2 -4310.097} C_VEL
LIN {X 0,Y 531.054,Z 239.838,A -85,B 0,C 180,E1 -4312.993,E2 -4312.993} C_VEL
LIN {X 0,Y 531.093,Z 239.831,A -85,B 0,C 180,E1 -4314.69,E2 -4314.69} C_VEL
LIN {X 0,Y 531.116,Z 239.822,A -85,B 0,C 180,E1 -4317.729,E2 -4317.729} C_VEL
LIN {X 0,Y 531.144,Z 239.828,A -85,B 0,C 180,E1 -4320.763,E2 -4320.763} C_VEL
LIN {X 0,Y 531.081,Z 239.83,A -85,B 0,C 180,E1 -4323.039,E2 -4323.039} C_VEL
LIN {X 0,Y 531.043,Z 239.833,A -85,B 0,C 180,E1 -4326.082,E2 -4326.082} C_VEL
LIN {X 0,Y 530.983,Z 239.845,A -85,B 0,C 180,E1 -4328.376,E2 -4328.376} C_VEL
LIN {X 0,Y 531.044,Z 239.831,A -85,B 0,C 180,E1 -4331.674,E2 -4331.674} C_VEL
LIN {X 0,Y 531.028,Z 239.834,A -85,B 0,C 180,E1 -4334.959,E2 -4334.959} C_VEL
LIN {X 0,Y 530.978,Z 239.84,A -85,B 0,C 180,E1 -4337.727,E2 -4337.727} C_VEL
LIN {X 0,Y 531.024,Z 239.84,A -85,B 0,C 180,E1 -4340.131,E2 -4340.131} C_VEL
LIN {X 0,Y 530.943,Z 239.847,A -85,B 0,C 180,E1 -4342.577,E2 -4342.577} C_VEL
LIN {X 0,Y 530.979,Z 239.839,A -85,B 0,C 180,E1 -4345.062,E2 -4345.062} C_VEL
LIN {X 0,Y 530.961,Z 239.844,A -85,B 0,C 180,E1 -4347.602,E2 -4347.602} C_VEL
LIN {X 0,Y 530.955,Z 239.848,A -85,B 0,C 180,E1 -4350.201,E2 -4350.201} C_VEL
LIN {X 0,Y 530.97,Z 239.84,A -85,B 0,C 180,E1 -4352.869,E2 -4352.869} C_VEL
LIN {X 0,Y 530.95,Z 239.848,A -85,B 0,C 180,E1 -4355.623,E2 -4355.623} C_VEL
LIN {X 0,Y 530.965,Z 239.844,A -85,B 0,C 180,E1 -4358.655,E2 -4358.655} C_VEL
LIN {X 0,Y 530.983,Z 239.847,A -85,B 0,C 180,E1 -4361.439,E2 -4361.439} C_VEL
LIN {X 0,Y 530.99,Z 239.948,A -85,B 0,C 180,E1 -4364.381,E2 -4364.381} C_VEL
LIN {X 0,Y 531.405,Z 243.048,A -85,B 0,C 180,E1 -4366.671,E2 -4366.671} C_VEL
LIN {X 0,Y 531.503,Z 246.335,A -85,B 0,C 180,E1 -4368.915,E2 -4368.915} C_VEL
LIN {X 0,Y 531.384,Z 250.534,A -85,B 0,C 180,E1 -4371.567,E2 -4371.567} C_VEL
LIN {X 0,Y 531.288,Z 255.315,A -85,B 0,C 180,E1 -4374.407,E2 -4374.407} C_VEL
LIN {X 0,Y 531.153,Z 260.224,A -85,B 0,C 180,E1 -4377.147,E2 -4377.147} C_VEL
LIN {X 0,Y 530.984,Z 265.238,A -85,B 0,C 180,E1 -4379.805,E2 -4379.805} C_VEL
LIN {X 0,Y 530.878,Z 270.561,A -85,B 0,C 180,E1 -4382.498,E2 -4382.498} C_VEL
LIN {X 0,Y 530.741,Z 275.54,A -85,B 0,C 180,E1 -4384.93,E2 -4384.93} C_VEL
LIN {X 0,Y 530.679,Z 282.015,A -85,B 0,C 180,E1 -4387.981,E2 -4387.981} C_VEL
LIN {X 0,Y 530.638,Z 287.897,A -85,B 0,C 180,E1 -4390.664,E2 -4390.664} C_VEL
LIN {X 0,Y 530.55,Z 293.352,A -85,B 0,C 180,E1 -4393.057,E2 -4393.057} C_VEL
LIN {X 0,Y 530.537,Z 298.76,A -85,B 0,C 180,E1 -4395.423,E2 -4395.423} C_VEL
LIN {X 0,Y 530.497,Z 301.39,A -85,B 0,C 180,E1 -4396.51,E2 -4396.51} C_VEL
LIN {X 0,Y 532.188,Z 311.543,A -85,B 0,C 180,E1 -4396.784,E2 -4396.784} C_VEL
LIN {X 0,Y 532.13,Z 320.647,A -85,B 0,C 180,E1 -4397.074,E2 -4397.074} C_VEL
LIN {X 0,Y 531.901,Z 331.011,A -85,B 0,C 180,E1 -4397.505,E2 -4397.505} C_VEL
LIN {X 0,Y 531.676,Z 340.624,A -85,B 0,C 180,E1 -4398.012,E2 -4398.012} C_VEL
LIN {X 0,Y 531.523,Z 349.149,A -85,B 0,C 180,E1 -4398.561,E2 -4398.561} C_VEL
LIN {X 0,Y 531.34,Z 357.881,A -85,B 0,C 180,E1 -4399.232,E2 -4399.232} C_VEL
LIN {X 0,Y 531.158,Z 365.278,A -85,B 0,C 180,E1 -4399.903,E2 -4399.903} C_VEL
LIN {X 0,Y 530.998,Z 372.499,A -85,B 0,C 180,E1 -4400.669,E2 -4400.669} C_VEL
LIN {X 0,Y 530.866,Z 378.702,A -85,B 0,C 180,E1 -4401.435,E2 -4401.435} C_VEL
LIN {X 0,Y 530.707,Z 385.238,A -85,B 0,C 180,E1 -4402.39,E2 -4402.39} C_VEL
LIN {X 0,Y 530.596,Z 391.111,A -85,B 0,C 180,E1 -4403.427,E2 -4403.427} C_VEL
LIN {X 0,Y 530.588,Z 395.228,A -85,B 0,C 180,E1 -4404.299,E2 -4404.299} C_VEL
LIN {X 0,Y 530.461,Z 399.546,A -85,B 0,C 180,E1 -4405.441,E2 -4405.441} C_VEL
LIN {X 0,Y 530.518,Z 401.911,A -85,B 0,C 180,E1 -4406.202,E2 -4406.202} C_VEL
LIN {X 0,Y 530.459,Z 403.705,A -85,B 0,C 180,E1 -4406.962,E2 -4406.962} C_VEL
LIN {X 0,Y 530.362,Z 406.141,A -85,B 0,C 180,E1 -4408.481,E2 -4408.481} C_VEL
LIN {X 0,Y 530.344,Z 406.728,A -85,B 0,C 180,E1 -4409.241,E2 -4409.241} C_VEL
LIN {X 0,Y 530.344,Z 406.728,A -85,B 0,C 180,E1 -4410.759,E2 -4410.759} C_VEL
LIN {X 0,Y 530.362,Z 406.141,A -85,B 0,C 180,E1 -4411.519,E2 -4411.519} C_VEL
LIN {X 0,Y 530.459,Z 403.705,A -85,B 0,C 180,E1 -4413.038,E2 -4413.038} C_VEL
LIN {X 0,Y 530.525,Z 400.763,A -85,B 0,C 180,E1 -4414.178,E2 -4414.178} C_VEL
LIN {X 0,Y 530.525,Z 396.779,A -85,B 0,C 180,E1 -4415.321,E2 -4415.321} C_VEL
LIN {X 0,Y 530.549,Z 392.471,A -85,B 0,C 180,E1 -4416.302,E2 -4416.302} C_VEL
LIN {X 0,Y 530.671,Z 387.549,A -85,B 0,C 180,E1 -4417.228,E2 -4417.228} C_VEL
LIN {X 0,Y 530.788,Z 381.454,A -85,B 0,C 180,E1 -4418.183,E2 -4418.183} C_VEL
LIN {X 0,Y 530.92,Z 375.754,A -85,B 0,C 180,E1 -4418.948,E2 -4418.948} C_VEL
LIN {X 0,Y 531.12,Z 367.198,A -85,B 0,C 180,E1 -4419.905,E2 -4419.905} C_VEL
LIN {X 0,Y 531.334,Z 359.016,A -85,B 0,C 180,E1 -4420.671,E2 -4420.671} C_VEL
LIN {X 0,Y 531.519,Z 350.502,A -85,B 0,C 180,E1 -4421.343,E2 -4421.343} C_VEL
LIN {X 0,Y 531.645,Z 341.958,A -85,B 0,C 180,E1 -4421.91,E2 -4421.91} C_VEL
LIN {X 0,Y 531.908,Z 332.02,A -85,B 0,C 180,E1 -4422.447,E2 -4422.447} C_VEL
LIN {X 0,Y 532.099,Z 323.224,A -85,B 0,C 180,E1 -4422.83,E2 -4422.83} C_VEL
LIN {X 0,Y 532.267,Z 313.295,A -85,B 0,C 180,E1 -4423.165,E2 -4423.165} C_VEL
LIN {X 0,Y 530.844,Z 303.733,A -85,B 0,C 180,E1 -4423.439,E2 -4423.439} C_VEL
LIN {X 0,Y 530.476,Z 301.229,A -85,B 0,C 180,E1 -4423.503,E2 -4423.503} C_VEL
LIN {X 0,Y 530.526,Z 295.157,A -85,B 0,C 180,E1 -4426.152,E2 -4426.152} C_VEL
LIN {X 0,Y 530.592,Z 289.722,A -85,B 0,C 180,E1 -4428.535,E2 -4428.535} C_VEL
LIN {X 0,Y 530.649,Z 284.326,A -85,B 0,C 180,E1 -4430.952,E2 -4430.952} C_VEL
LIN {X 0,Y 530.721,Z 277.825,A -85,B 0,C 180,E1 -4433.972,E2 -4433.972} C_VEL
LIN {X 0,Y 530.846,Z 272.048,A -85,B 0,C 180,E1 -4436.752,E2 -4436.752} C_VEL
LIN {X 0,Y 530.946,Z 266.923,A -85,B 0,C 180,E1 -4439.324,E2 -4439.324} C_VEL
LIN {X 0,Y 531.098,Z 261.561,A -85,B 0,C 180,E1 -4442.12,E2 -4442.12} C_VEL
LIN {X 0,Y 531.272,Z 256.533,A -85,B 0,C 180,E1 -4444.895,E2 -4444.895} C_VEL
LIN {X 0,Y 531.378,Z 252.082,A -85,B 0,C 180,E1 -4447.478,E2 -4447.478} C_VEL
LIN {X 0,Y 531.484,Z 247.409,A -85,B 0,C 180,E1 -4450.386,E2 -4450.386} C_VEL
LIN {X 0,Y 531.481,Z 244.354,A -85,B 0,C 180,E1 -4452.406,E2 -4452.406} C_VEL
LIN {X 0,Y 531.171,Z 241.404,A -85,B 0,C 180,E1 -4454.526,E2 -4454.526} C_VEL
LIN {X 0,Y 530.989,Z 239.95,A -85,B 0,C 180,E1 -4455.619,E2 -4455.619} C_VEL
LIN {X 0,Y 530.983,Z 239.846,A -85,B 0,C 180,E1 -4458.561,E2 -4458.561} C_VEL
LIN {X 0,Y 530.955,Z 239.846,A -85,B 0,C 180,E1 -4461.526,E2 -4461.526} C_VEL
LIN {X 0,Y 530.95,Z 239.85,A -85,B 0,C 180,E1 -4464.377,E2 -4464.377} C_VEL
LIN {X 0,Y 530.97,Z 239.84,A -85,B 0,C 180,E1 -4467.131,E2 -4467.131} C_VEL
LIN {X 0,Y 530.955,Z 239.848,A -85,B 0,C 180,E1 -4469.799,E2 -4469.799} C_VEL
LIN {X 0,Y 530.963,Z 239.843,A -85,B 0,C 180,E1 -4472.475,E2 -4472.475} C_VEL
LIN {X 0,Y 530.979,Z 239.839,A -85,B 0,C 180,E1 -4474.938,E2 -4474.938} C_VEL
LIN {X 0,Y 530.97,Z 239.843,A -85,B 0,C 180,E1 -4478.243,E2 -4478.243} C_VEL
LIN {X 0,Y 530.98,Z 239.839,A -85,B 0,C 180,E1 -4480.673,E2 -4480.673} C_VEL
LIN {X 0,Y 530.96,Z 239.843,A -85,B 0,C 180,E1 -4483.067,E2 -4483.067} C_VEL
LIN {X 0,Y 531.015,Z 239.841,A -85,B 0,C 180,E1 -4485.432,E2 -4485.432} C_VEL
LIN {X 0,Y 531.029,Z 239.833,A -85,B 0,C 180,E1 -4488.546,E2 -4488.546} C_VEL
LIN {X 0,Y 530.983,Z 239.845,A -85,B 0,C 180,E1 -4491.624,E2 -4491.624} C_VEL
LIN {X 0,Y 531.043,Z 239.833,A -85,B 0,C 180,E1 -4493.918,E2 -4493.918} C_VEL
LIN {X 0,Y 531.081,Z 239.83,A -85,B 0,C 180,E1 -4496.961,E2 -4496.961} C_VEL
LIN {X 0,Y 531.123,Z 239.821,A -85,B 0,C 180,E1 -4499.996,E2 -4499.996} C_VEL
LIN {X 0,Y 531.087,Z 239.832,A -85,B 0,C 180,E1 -4503.03,E2 -4503.03} C_VEL
LIN {X 0,Y 531.034,Z 239.832,A -85,B 0,C 180,E1 -4506.073,E2 -4506.073} C_VEL
LIN {X 0,Y 530.994,Z 239.844,A -85,B 0,C 180,E1 -4509.134,E2 -4509.134} C_VEL
LIN {X 0,Y 531.037,Z 239.832,A -85,B 0,C 180,E1 -4511.671,E2 -4511.671} C_VEL
LIN {X 0,Y 531.007,Z 239.843,A -85,B 0,C 180,E1 -4514.951,E2 -4514.951} C_VEL
LIN {X 0,Y 530.955,Z 239.842,A -85,B 0,C 180,E1 -4517.719,E2 -4517.719} C_VEL
LIN {X 0,Y 530.997,Z 239.838,A -85,B 0,C 180,E1 -4520.122,E2 -4520.122} C_VEL
LIN {X 0,Y 530.915,Z 239.854,A -85,B 0,C 180,E1 -4522.568,E2 -4522.568} C_VEL
LIN {X 0,Y 530.972,Z 239.843,A -85,B 0,C 180,E1 -4525.053,E2 -4525.053} C_VEL
LIN {X 0,Y 530.982,Z 239.838,A -85,B 0,C 180,E1 -4527.59,E2 -4527.59} C_VEL
LIN {X 0,Y 530.935,Z 239.851,A -85,B 0,C 180,E1 -4530.64,E2 -4530.64} C_VEL
LIN {X 0,Y 530.952,Z 239.843,A -85,B 0,C 180,E1 -4533.768,E2 -4533.768} C_VEL
LIN {X 0,Y 530.927,Z 239.851,A -85,B 0,C 180,E1 -4536.553,E2 -4536.553} C_VEL
LIN {X 0,Y 530.96,Z 239.845,A -85,B 0,C 180,E1 -4539.853,E2 -4539.853} C_VEL
LIN {X 0,Y 530.942,Z 239.848,A -85,B 0,C 180,E1 -4542.451,E2 -4542.451} C_VEL
LIN {X 0,Y 530.948,Z 239.844,A -85,B 0,C 180,E1 -4543.539,E2 -4543.539} C_VEL
LIN {X 0,Y 530.258,Z 239.937,A -85,B 0,C 180,E1 -4544.172,E2 -4544.172} C_VEL
LIN {X 0,Y 527.397,Z 240.287,A -85,B 0,C 180,E1 -4545.201,E2 -4545.201} C_VEL
LIN {X 0,Y 524.991,Z 240.593,A -85,B 0,C 180,E1 -4546.029,E2 -4546.029} C_VEL
LIN {X 0,Y 523.957,Z 240.715,A -85,B 0,C 180,E1 -4546.668,E2 -4546.668} C_VEL
LIN {X 0,Y 523.872,Z 240.724,A -85,B 0,C 180,E1 -4546.885,E2 -4546.885} C_VEL
LIN {X 0,Y 523.961,Z 240.721,A -85,B 0,C 180,E1 -4549.923,E2 -4549.923} C_VEL
LIN {X 0,Y 523.855,Z 240.726,A -85,B 0,C 180,E1 -4552.865,E2 -4552.865} C_VEL
LIN {X 0,Y 523.888,Z 240.729,A -85,B 0,C 180,E1 -4555.707,E2 -4555.707} C_VEL
LIN {X 0,Y 523.873,Z 240.725,A -85,B 0,C 180,E1 -4558.454,E2 -4558.454} C_VEL
LIN {X 0,Y 523.898,Z 240.722,A -85,B 0,C 180,E1 -4561.124,E2 -4561.124} C_VEL
LIN {X 0,Y 523.928,Z 240.721,A -85,B 0,C 180,E1 -4563.976,E2 -4563.976} C_VEL
LIN {X 0,Y 523.908,Z 240.721,A -85,B 0,C 180,E1 -4566.27,E2 -4566.27} C_VEL
LIN {X 0,Y 523.894,Z 240.722,A -85,B 0,C 180,E1 -4568.765,E2 -4568.765} C_VEL
LIN {X 0,Y 523.894,Z 240.727,A -85,B 0,C 180,E1 -4571.219,E2 -4571.219} C_VEL
LIN {X 0,Y 523.896,Z 240.728,A -85,B 0,C 180,E1 -4573.638,E2 -4573.638} C_VEL
LIN {X 0,Y 523.887,Z 240.725,A -85,B 0,C 180,E1 -4576.027,E2 -4576.027} C_VEL
LIN {X 0,Y 523.945,Z 240.716,A -85,B 0,C 180,E1 -4578.393,E2 -4578.393} C_VEL
LIN {X 0,Y 523.945,Z 240.721,A -85,B 0,C 180,E1 -4581.515,E2 -4581.515} C_VEL
LIN {X 0,Y 523.986,Z 240.713,A -85,B 0,C 180,E1 -4583.84,E2 -4583.84} C_VEL
LIN {X 0,Y 524.015,Z 240.714,A -85,B 0,C 180,E1 -4586.925,E2 -4586.925} C_VEL
LIN {X 0,Y 524.041,Z 240.706,A -85,B 0,C 180,E1 -4590,E2 -4590} C_VEL
LIN {X 0,Y 524.015,Z 240.714,A -85,B 0,C 180,E1 -4593.075,E2 -4593.075} C_VEL
LIN {X 0,Y 523.986,Z 240.713,A -85,B 0,C 180,E1 -4596.16,E2 -4596.16} C_VEL
LIN {X 0,Y 523.945,Z 240.721,A -85,B 0,C 180,E1 -4598.485,E2 -4598.485} C_VEL
LIN {X 0,Y 523.955,Z 240.715,A -85,B 0,C 180,E1 -4601.753,E2 -4601.753} C_VEL
LIN {X 0,Y 523.939,Z 240.721,A -85,B 0,C 180,E1 -4605.06,E2 -4605.06} C_VEL
LIN {X 0,Y 523.905,Z 240.723,A -85,B 0,C 180,E1 -4607.971,E2 -4607.971} C_VEL
LIN {X 0,Y 523.908,Z 240.728,A -85,B 0,C 180,E1 -4610.412,E2 -4610.412} C_VEL
LIN {X 0,Y 523.901,Z 240.723,A -85,B 0,C 180,E1 -4612.893,E2 -4612.893} C_VEL
LIN {X 0,Y 523.921,Z 240.718,A -85,B 0,C 180,E1 -4615.42,E2 -4615.42} C_VEL
LIN {X 0,Y 523.911,Z 240.724,A -85,B 0,C 180,E1 -4618.002,E2 -4618.002} C_VEL
LIN {X 0,Y 523.892,Z 240.723,A -85,B 0,C 180,E1 -4620.86,E2 -4620.86} C_VEL
LIN {X 0,Y 523.904,Z 240.723,A -85,B 0,C 180,E1 -4623.739,E2 -4623.739} C_VEL
LIN {X 0,Y 523.866,Z 240.729,A -85,B 0,C 180,E1 -4626.408,E2 -4626.408} C_VEL
LIN {X 0,Y 523.92,Z 240.718,A -85,B 0,C 180,E1 -4629.084,E2 -4629.084} C_VEL
LIN {X 0,Y 523.928,Z 240.718,A -85,B 0,C 180,E1 -4631.318,E2 -4631.318} C_VEL
LIN {X 0,Y 523.911,Z 240.72,A -85,B 0,C 180,E1 -4634.696,E2 -4634.696} C_VEL
LIN {X 0,Y 523.919,Z 240.726,A -85,B 0,C 180,E1 -4637.887,E2 -4637.887} C_VEL
LIN {X 0,Y 523.886,Z 240.723,A -85,B 0,C 180,E1 -4640.921,E2 -4640.921} C_VEL
LIN {X 0,Y 523.887,Z 240.729,A -85,B 0,C 180,E1 -4643.832,E2 -4643.832} C_VEL
LIN {X 0,Y 523.903,Z 240.72,A -85,B 0,C 180,E1 -4646.641,E2 -4646.641} C_VEL
LIN {X 0,Y 523.917,Z 240.725,A -85,B 0,C 180,E1 -4649.361,E2 -4649.361} C_VEL
LIN {X 0,Y 523.944,Z 240.715,A -85,B 0,C 180,E1 -4652.286,E2 -4652.286} C_VEL
LIN {X 0,Y 523.919,Z 240.719,A -85,B 0,C 180,E1 -4654.586,E2 -4654.586} C_VEL
LIN {X 0,Y 523.88,Z 240.729,A -85,B 0,C 180,E1 -4657.111,E2 -4657.111} C_VEL
LIN {X 0,Y 523.951,Z 240.716,A -85,B 0,C 180,E1 -4659.871,E2 -4659.871} C_VEL
LIN {X 0,Y 523.931,Z 240.721,A -85,B 0,C 180,E1 -4662.842,E2 -4662.842} C_VEL
LIN {X 0,Y 523.953,Z 240.722,A -85,B 0,C 180,E1 -4665.241,E2 -4665.241} C_VEL
LIN {X 0,Y 523.992,Z 240.71,A -85,B 0,C 180,E1 -4668.399,E2 -4668.399} C_VEL
LIN {X 0,Y 523.967,Z 240.714,A -85,B 0,C 180,E1 -4671.52,E2 -4671.52} C_VEL
LIN {X 0,Y 523.999,Z 240.708,A -85,B 0,C 180,E1 -4673.845,E2 -4673.845} C_VEL
LIN {X 0,Y 524.055,Z 240.709,A -85,B 0,C 180,E1 -4676.93,E2 -4676.93} C_VEL
LIN {X 0,Y 524.094,Z 240.697,A -85,B 0,C 180,E1 -4680.004,E2 -4680.004} C_VEL
LIN {X 0,Y 524.022,Z 240.709,A -85,B 0,C 180,E1 -4683.08,E2 -4683.08} C_VEL
LIN {X 0,Y 524.009,Z 240.71,A -85,B 0,C 180,E1 -4686.164,E2 -4686.164} C_VEL
LIN {X 0,Y 523.973,Z 240.712,A -85,B 0,C 180,E1 -4689.266,E2 -4689.266} C_VEL
LIN {X 0,Y 523.993,Z 240.71,A -85,B 0,C 180,E1 -4691.74,E2 -4691.74} C_VEL
LIN {X 0,Y 523.99,Z 240.71,A -85,B 0,C 180,E1 -4695.056,E2 -4695.056} C_VEL
LIN {X 0,Y 523.942,Z 240.719,A -85,B 0,C 180,E1 -4697.973,E2 -4697.973} C_VEL
LIN {X 0,Y 523.971,Z 240.719,A -85,B 0,C 180,E1 -4700.414,E2 -4700.414} C_VEL
LIN {X 0,Y 523.909,Z 240.72,A -85,B 0,C 180,E1 -4702.897,E2 -4702.897} C_VEL
LIN {X 0,Y 523.92,Z 240.719,A -85,B 0,C 180,E1 -4705.424,E2 -4705.424} C_VEL
LIN {X 0,Y 523.913,Z 240.727,A -85,B 0,C 180,E1 -4708.005,E2 -4708.005} C_VEL
LIN {X 0,Y 523.937,Z 240.716,A -85,B 0,C 180,E1 -4710.856,E2 -4710.856} C_VEL
LIN {X 0,Y 523.943,Z 240.721,A -85,B 0,C 180,E1 -4713.734,E2 -4713.734} C_VEL
LIN {X 0,Y 523.9,Z 240.725,A -85,B 0,C 180,E1 -4716.403,E2 -4716.403} C_VEL
LIN {X 0,Y 523.915,Z 240.723,A -85,B 0,C 180,E1 -4719.088,E2 -4719.088} C_VEL
LIN {X 0,Y 523.942,Z 240.723,A -85,B 0,C 180,E1 -4722.123,E2 -4722.123} C_VEL
LIN {X 0,Y 523.961,Z 240.978,A -85,B 0,C 180,E1 -4724.229,E2 -4724.229} C_VEL
LIN {X 0,Y 524.419,Z 244.556,A -85,B 0,C 180,E1 -4726.885,E2 -4726.885} C_VEL
LIN {X 0,Y 524.509,Z 247.557,A -85,B 0,C 180,E1 -4728.963,E2 -4728.963} C_VEL
LIN {X 0,Y 524.356,Z 252.237,A -85,B 0,C 180,E1 -4731.937,E2 -4731.937} C_VEL
LIN {X 0,Y 524.267,Z 257.121,A -85,B 0,C 180,E1 -4734.861,E2 -4734.861} C_VEL
LIN {X 0,Y 524.089,Z 262.117,A -85,B 0,C 180,E1 -4737.656,E2 -4737.656} C_VEL
LIN {X 0,Y 523.897,Z 267.825,A -85,B 0,C 180,E1 -4740.691,E2 -4740.691} C_VEL
LIN {X 0,Y 523.791,Z 272.054,A -85,B 0,C 180,E1 -4742.859,E2 -4742.859} C_VEL
LIN {X 0,Y 523.667,Z 278.193,A -85,B 0,C 180,E1 -4745.872,E2 -4745.872} C_VEL
LIN {X 0,Y 523.569,Z 284.262,A -85,B 0,C 180,E1 -4748.751,E2 -4748.751} C_VEL
LIN {X 0,Y 523.529,Z 289.579,A -85,B 0,C 180,E1 -4751.206,E2 -4751.206} C_VEL
LIN {X 0,Y 523.431,Z 294.97,A -85,B 0,C 180,E1 -4753.623,E2 -4753.623} C_VEL
LIN {X 0,Y 523.418,Z 301.045,A -85,B 0,C 180,E1 -4756.311,E2 -4756.311} C_VEL
LIN {X 0,Y 525.334,Z 313.974,A -85,B 0,C 180,E1 -4756.682,E2 -4756.682} C_VEL
LIN {X 0,Y 525.032,Z 327.794,A -85,B 0,C 180,E1 -4757.191,E2 -4757.191} C_VEL
LIN {X 0,Y 524.787,Z 338.938,A -85,B 0,C 180,E1 -4757.763,E2 -4757.763} C_VEL
LIN {X 0,Y 524.591,Z 347.944,A -85,B 0,C 180,E1 -4758.334,E2 -4758.334} C_VEL
LIN {X 0,Y 524.341,Z 356.549,A -85,B 0,C 180,E1 -4758.989,E2 -4758.989} C_VEL
LIN {X 0,Y 524.137,Z 365.082,A -85,B 0,C 180,E1 -4759.766,E2 -4759.766} C_VEL
LIN {X 0,Y 523.969,Z 372.304,A -85,B 0,C 180,E1 -4760.543,E2 -4760.543} C_VEL
LIN {X 0,Y 523.794,Z 378.506,A -85,B 0,C 180,E1 -4761.318,E2 -4761.318} C_VEL
LIN {X 0,Y 523.653,Z 385.043,A -85,B 0,C 180,E1 -4762.287,E2 -4762.287} C_VEL
LIN {X 0,Y 523.58,Z 389.544,A -85,B 0,C 180,E1 -4763.062,E2 -4763.062} C_VEL
LIN {X 0,Y 523.505,Z 395.033,A -85,B 0,C 180,E1 -4764.221,E2 -4764.221} C_VEL
LIN {X 0,Y 523.366,Z 399.351,A -85,B 0,C 180,E1 -4765.379,E2 -4765.379} C_VEL
LIN {X 0,Y 523.445,Z 401.717,A -85,B 0,C 180,E1 -4766.151,E2 -4766.151} C_VEL
LIN {X 0,Y 523.369,Z 403.51,A -85,B 0,C 180,E1 -4766.921,E2 -4766.921} C_VEL
LIN {X 0,Y 523.276,Z 405.947,A -85,B 0,C 180,E1 -4768.461,E2 -4768.461} C_VEL
LIN {X 0,Y 523.251,Z 406.533,A -85,B 0,C 180,E1 -4769.23,E2 -4769.23} C_VEL
LIN {X 0,Y 523.251,Z 406.533,A -85,B 0,C 180,E1 -4770.77,E2 -4770.77} C_VEL
LIN {X 0,Y 523.276,Z 405.947,A -85,B 0,C 180,E1 -4771.539,E2 -4771.539} C_VEL
LIN {X 0,Y 523.369,Z 403.51,A -85,B 0,C 180,E1 -4773.079,E2 -4773.079} C_VEL
LIN {X 0,Y 523.428,Z 400.568,A -85,B 0,C 180,E1 -4774.235,E2 -4774.235} C_VEL
LIN {X 0,Y 523.461,Z 396.585,A -85,B 0,C 180,E1 -4775.393,E2 -4775.393} C_VEL
LIN {X 0,Y 523.518,Z 391.374,A -85,B 0,C 180,E1 -4776.569,E2 -4776.569} C_VEL
LIN {X 0,Y 523.611,Z 386.198,A -85,B 0,C 180,E1 -4777.519,E2 -4777.519} C_VEL
LIN {X 0,Y 523.766,Z 379.882,A -85,B 0,C 180,E1 -4778.488,E2 -4778.488} C_VEL
LIN {X 0,Y 523.923,Z 373.931,A -85,B 0,C 180,E1 -4779.263,E2 -4779.263} C_VEL
LIN {X 0,Y 524.08,Z 367.002,A -85,B 0,C 180,E1 -4780.04,E2 -4780.04} C_VEL
LIN {X 0,Y 524.319,Z 358.821,A -85,B 0,C 180,E1 -4780.816,E2 -4780.816} C_VEL
LIN {X 0,Y 524.532,Z 350.306,A -85,B 0,C 180,E1 -4781.496,E2 -4781.496} C_VEL
LIN {X 0,Y 524.659,Z 341.707,A -85,B 0,C 180,E1 -4782.074,E2 -4782.074} C_VEL
LIN {X 0,Y 524.947,Z 331.824,A -85,B 0,C 180,E1 -4782.614,E2 -4782.614} C_VEL
LIN {X 0,Y 525.166,Z 323.029,A -85,B 0,C 180,E1 -4783.002,E2 -4783.002} C_VEL
LIN {X 0,Y 525.298,Z 312.661,A -85,B 0,C 180,E1 -4783.356,E2 -4783.356} C_VEL
LIN {X 0,Y 523.553,Z 302.361,A -85,B 0,C 180,E1 -4783.651,E2 -4783.651} C_VEL
LIN {X 0,Y 523.418,Z 301.045,A -85,B 0,C 180,E1 -4783.689,E2 -4783.689} C_VEL
LIN {X 0,Y 523.431,Z 294.97,A -85,B 0,C 180,E1 -4786.377,E2 -4786.377} C_VEL
LIN {X 0,Y 523.529,Z 289.574,A -85,B 0,C 180,E1 -4788.794,E2 -4788.794} C_VEL
LIN {X 0,Y 523.568,Z 284.247,A -85,B 0,C 180,E1 -4791.249,E2 -4791.249} C_VEL
LIN {X 0,Y 523.667,Z 278.169,A -85,B 0,C 180,E1 -4794.128,E2 -4794.128} C_VEL
LIN {X 0,Y 523.785,Z 272.051,A -85,B 0,C 180,E1 -4797.142,E2 -4797.142} C_VEL
LIN {X 0,Y 523.912,Z 266.926,A -85,B 0,C 180,E1 -4799.757,E2 -4799.757} C_VEL
LIN {X 0,Y 524.093,Z 261.914,A -85,B 0,C 180,E1 -4802.438,E2 -4802.438} C_VEL
LIN {X 0,Y 524.249,Z 257.006,A -85,B 0,C 180,E1 -4805.2,E2 -4805.2} C_VEL
LIN {X 0,Y 524.358,Z 252.206,A -85,B 0,C 180,E1 -4808.063,E2 -4808.063} C_VEL
LIN {X 0,Y 524.508,Z 247.546,A -85,B 0,C 180,E1 -4811.037,E2 -4811.037} C_VEL
LIN {X 0,Y 524.335,Z 243.806,A -85,B 0,C 180,E1 -4813.628,E2 -4813.628} C_VEL
LIN {X 0,Y 523.96,Z 240.978,A -85,B 0,C 180,E1 -4815.771,E2 -4815.771} C_VEL
LIN {X 0,Y 523.942,Z 240.722,A -85,B 0,C 180,E1 -4817.877,E2 -4817.877} C_VEL
LIN {X 0,Y 523.915,Z 240.722,A -85,B 0,C 180,E1 -4821.079,E2 -4821.079} C_VEL
LIN {X 0,Y 523.897,Z 240.728,A -85,B 0,C 180,E1 -4823.822,E2 -4823.822} C_VEL
LIN {X 0,Y 523.929,Z 240.719,A -85,B 0,C 180,E1 -4826.632,E2 -4826.632} C_VEL
LIN {X 0,Y 523.946,Z 240.716,A -85,B 0,C 180,E1 -4829.352,E2 -4829.352} C_VEL
LIN {X 0,Y 523.921,Z 240.722,A -85,B 0,C 180,E1 -4832.291,E2 -4832.291} C_VEL
LIN {X 0,Y 523.92,Z 240.719,A -85,B 0,C 180,E1 -4834.576,E2 -4834.576} C_VEL
LIN {X 0,Y 523.909,Z 240.72,A -85,B 0,C 180,E1 -4837.103,E2 -4837.103} C_VEL
LIN {X 0,Y 523.978,Z 240.718,A -85,B 0,C 180,E1 -4839.863,E2 -4839.863} C_VEL
LIN {X 0,Y 523.94,Z 240.716,A -85,B 0,C 180,E1 -4842.833,E2 -4842.833} C_VEL
LIN {X 0,Y 523.973,Z 240.715,A -85,B 0,C 180,E1 -4845.232,E2 -4845.232} C_VEL
LIN {X 0,Y 524.009,Z 240.707,A -85,B 0,C 180,E1 -4848.39,E2 -4848.39} C_VEL
LIN {X 0,Y 523.947,Z 240.723,A -85,B 0,C 180,E1 -4851.511,E2 -4851.511} C_VEL
LIN {X 0,Y 524.009,Z 240.71,A -85,B 0,C 180,E1 -4853.836,E2 -4853.836} C_VEL
LIN {X 0,Y 524.022,Z 240.709,A -85,B 0,C 180,E1 -4856.92,E2 -4856.92} C_VEL
LIN {X 0,Y 524.094,Z 240.697,A -85,B 0,C 180,E1 -4859.996,E2 -4859.996} C_VEL
LIN {X 0,Y 524.055,Z 240.709,A -85,B 0,C 180,E1 -4863.07,E2 -4863.07} C_VEL
LIN {X 0,Y 523.999,Z 240.708,A -85,B 0,C 180,E1 -4866.155,E2 -4866.155} C_VEL
LIN {X 0,Y 523.965,Z 240.718,A -85,B 0,C 180,E1 -4869.257,E2 -4869.257} C_VEL
LIN {X 0,Y 523.988,Z 240.71,A -85,B 0,C 180,E1 -4871.737,E2 -4871.737} C_VEL
LIN {X 0,Y 523.969,Z 240.718,A -85,B 0,C 180,E1 -4875.047,E2 -4875.047} C_VEL
LIN {X 0,Y 523.922,Z 240.718,A -85,B 0,C 180,E1 -4877.965,E2 -4877.965} C_VEL
LIN {X 0,Y 523.945,Z 240.719,A -85,B 0,C 180,E1 -4880.405,E2 -4880.405} C_VEL
LIN {X 0,Y 523.88,Z 240.729,A -85,B 0,C 180,E1 -4882.889,E2 -4882.889} C_VEL
LIN {X 0,Y 523.919,Z 240.719,A -85,B 0,C 180,E1 -4885.414,E2 -4885.414} C_VEL
LIN {X 0,Y 523.935,Z 240.718,A -85,B 0,C 180,E1 -4887.994,E2 -4887.994} C_VEL
LIN {X 0,Y 523.906,Z 240.723,A -85,B 0,C 180,E1 -4890.85,E2 -4890.85} C_VEL
LIN {X 0,Y 523.922,Z 240.719,A -85,B 0,C 180,E1 -4893.73,E2 -4893.73} C_VEL
LIN {X 0,Y 523.882,Z 240.731,A -85,B 0,C 180,E1 -4896.4,E2 -4896.4} C_VEL
LIN {X 0,Y 523.886,Z 240.723,A -85,B 0,C 180,E1 -4899.079,E2 -4899.079} C_VEL
LIN {X 0,Y 523.919,Z 240.726,A -85,B 0,C 180,E1 -4902.113,E2 -4902.113} C_VEL
LIN {X 0,Y 523.911,Z 240.72,A -85,B 0,C 180,E1 -4905.304,E2 -4905.304} C_VEL
LIN {X 0,Y 523.872,Z 240.724,A -85,B 0,C 180,E1 -4906.885,E2 -4906.885} C_VEL
LIN {X 0,Y 523.2,Z 240.811,A -85,B 0,C 180,E1 -4907.526,E2 -4907.526} C_VEL
LIN {X 0,Y 520.344,Z 241.166,A -85,B 0,C 180,E1 -4908.568,E2 -4908.568} C_VEL
LIN {X 0,Y 517.95,Z 241.463,A -85,B 0,C 180,E1 -4909.407,E2 -4909.407} C_VEL
LIN {X 0,Y 516.949,Z 241.595,A -85,B 0,C 180,E1 -4910.055,E2 -4910.055} C_VEL
LIN {X 0,Y 516.881,Z 241.6,A -85,B 0,C 180,E1 -4910.274,E2 -4910.274} C_VEL
LIN {X 0,Y 516.828,Z 241.603,A -85,B 0,C 180,E1 -4913.338,E2 -4913.338} C_VEL
LIN {X 0,Y 516.855,Z 241.603,A -85,B 0,C 180,E1 -4916.118,E2 -4916.118} C_VEL
LIN {X 0,Y 516.834,Z 241.601,A -85,B 0,C 180,E1 -4918.932,E2 -4918.932} C_VEL
LIN {X 0,Y 516.867,Z 241.604,A -85,B 0,C 180,E1 -4921.582,E2 -4921.582} C_VEL
LIN {X 0,Y 516.883,Z 241.596,A -85,B 0,C 180,E1 -4924.209,E2 -4924.209} C_VEL
LIN {X 0,Y 516.847,Z 241.6,A -85,B 0,C 180,E1 -4926.776,E2 -4926.776} C_VEL
LIN {X 0,Y 516.873,Z 241.603,A -85,B 0,C 180,E1 -4929.729,E2 -4929.729} C_VEL
LIN {X 0,Y 516.877,Z 241.598,A -85,B 0,C 180,E1 -4932.595,E2 -4932.595} C_VEL
LIN {X 0,Y 516.897,Z 241.599,A -85,B 0,C 180,E1 -4935.029,E2 -4935.029} C_VEL
LIN {X 0,Y 516.935,Z 241.59,A -85,B 0,C 180,E1 -4938.233,E2 -4938.233} C_VEL
LIN {X 0,Y 516.909,Z 241.599,A -85,B 0,C 180,E1 -4941.399,E2 -4941.399} C_VEL
LIN {X 0,Y 516.954,Z 241.59,A -85,B 0,C 180,E1 -4943.756,E2 -4943.756} C_VEL
LIN {X 0,Y 516.981,Z 241.59,A -85,B 0,C 180,E1 -4946.883,E2 -4946.883} C_VEL
LIN {X 0,Y 517.012,Z 241.581,A -85,B 0,C 180,E1 -4950,E2 -4950} C_VEL
LIN {X 0,Y 516.981,Z 241.59,A -85,B 0,C 180,E1 -4953.117,E2 -4953.117} C_VEL
LIN {X 0,Y 516.954,Z 241.59,A -85,B 0,C 180,E1 -4956.244,E2 -4956.244} C_VEL
LIN {X 0,Y 516.909,Z 241.599,A -85,B 0,C 180,E1 -4958.601,E2 -4958.601} C_VEL
LIN {X 0,Y 516.914,Z 241.592,A -85,B 0,C 180,E1 -4961.825,E2 -4961.825} C_VEL
LIN {X 0,Y 516.89,Z 241.598,A -85,B 0,C 180,E1 -4965.154,E2 -4965.154} C_VEL
LIN {X 0,Y 516.864,Z 241.603,A -85,B 0,C 180,E1 -4968.224,E2 -4968.224} C_VEL
LIN {X 0,Y 516.852,Z 241.604,A -85,B 0,C 180,E1 -4970.703,E2 -4970.703} C_VEL
LIN {X 0,Y 516.847,Z 241.6,A -85,B 0,C 180,E1 -4973.224,E2 -4973.224} C_VEL
LIN {X 0,Y 516.886,Z 241.601,A -85,B 0,C 180,E1 -4976.2,E2 -4976.2} C_VEL
LIN {X 0,Y 516.882,Z 241.595,A -85,B 0,C 180,E1 -4979.306,E2 -4979.306} C_VEL
LIN {X 0,Y 516.842,Z 241.604,A -85,B 0,C 180,E1 -4982.548,E2 -4982.548} C_VEL
LIN {X 0,Y 516.826,Z 241.602,A -85,B 0,C 180,E1 -4985.336,E2 -4985.336} C_VEL
LIN {X 0,Y 516.831,Z 241.609,A -85,B 0,C 180,E1 -4987.948,E2 -4987.948} C_VEL
LIN {X 0,Y 516.865,Z 241.598,A -85,B 0,C 180,E1 -4990.742,E2 -4990.742} C_VEL
LIN {X 0,Y 516.833,Z 241.61,A -85,B 0,C 180,E1 -4993.907,E2 -4993.907} C_VEL
LIN {X 0,Y 516.878,Z 241.601,A -85,B 0,C 180,E1 -4996.106,E2 -4996.106} C_VEL
LIN {X 0,Y 516.862,Z 241.6,A -85,B 0,C 180,E1 -4999.265,E2 -4999.265} C_VEL
LIN {X 0,Y 516.821,Z 241.604,A -85,B 0,C 180,E1 -5002.279,E2 -5002.279} C_VEL
LIN {X 0,Y 516.855,Z 241.601,A -85,B 0,C 180,E1 -5005.181,E2 -5005.181} C_VEL
LIN {X 0,Y 516.837,Z 241.604,A -85,B 0,C 180,E1 -5007.98,E2 -5007.98} C_VEL
LIN {X 0,Y 516.886,Z 241.595,A -85,B 0,C 180,E1 -5010.7,E2 -5010.7} C_VEL
LIN {X 0,Y 516.909,Z 241.595,A -85,B 0,C 180,E1 -5013.809,E2 -5013.809} C_VEL
LIN {X 0,Y 516.834,Z 241.603,A -85,B 0,C 180,E1 -5016.781,E2 -5016.781} C_VEL
LIN {X 0,Y 516.912,Z 241.594,A -85,B 0,C 180,E1 -5019.737,E2 -5019.737} C_VEL
LIN {X 0,Y 516.881,Z 241.597,A -85,B 0,C 180,E1 -5022.6,E2 -5022.6} C_VEL
LIN {X 0,Y 516.918,Z 241.598,A -85,B 0,C 180,E1 -5025.035,E2 -5025.035} C_VEL
LIN {X 0,Y 516.945,Z 241.587,A -85,B 0,C 180,E1 -5028.239,E2 -5028.239} C_VEL
LIN {X 0,Y 516.935,Z 241.591,A -85,B 0,C 180,E1 -5031.404,E2 -5031.404} C_VEL
LIN {X 0,Y 516.968,Z 241.584,A -85,B 0,C 180,E1 -5033.761,E2 -5033.761} C_VEL
LIN {X 0,Y 516.996,Z 241.589,A -85,B 0,C 180,E1 -5036.888,E2 -5036.888} C_VEL
LIN {X 0,Y 517.066,Z 241.572,A -85,B 0,C 180,E1 -5040.005,E2 -5040.005} C_VEL
LIN {X 0,Y 517.064,Z 241.576,A -85,B 0,C 180,E1 -5042.341,E2 -5042.341} C_VEL
LIN {X 0,Y 517.007,Z 241.579,A -85,B 0,C 180,E1 -5045.464,E2 -5045.464} C_VEL
LIN {X 0,Y 516.946,Z 241.588,A -85,B 0,C 180,E1 -5047.818,E2 -5047.818} C_VEL
LIN {X 0,Y 516.942,Z 241.59,A -85,B 0,C 180,E1 -5050.976,E2 -5050.976} C_VEL
LIN {X 0,Y 516.886,Z 241.6,A -85,B 0,C 180,E1 -5054.17,E2 -5054.17} C_VEL
LIN {X 0,Y 516.894,Z 241.599,A -85,B 0,C 180,E1 -5056.594,E2 -5056.594} C_VEL
LIN {X 0,Y 516.889,Z 241.595,A -85,B 0,C 180,E1 -5059.049,E2 -5059.049} C_VEL
LIN {X 0,Y 516.884,Z 241.596,A -85,B 0,C 180,E1 -5061.541,E2 -5061.541} C_VEL
LIN {X 0,Y 516.882,Z 241.601,A -85,B 0,C 180,E1 -5064.36,E2 -5064.36} C_VEL
LIN {X 0,Y 516.858,Z 241.6,A -85,B 0,C 180,E1 -5066.665,E2 -5066.665} C_VEL
LIN {X 0,Y 516.909,Z 241.594,A -85,B 0,C 180,E1 -5069.526,E2 -5069.526} C_VEL
LIN {X 0,Y 516.898,Z 241.594,A -85,B 0,C 180,E1 -5072.546,E2 -5072.546} C_VEL
LIN {X 0,Y 516.864,Z 241.599,A -85,B 0,C 180,E1 -5075.331,E2 -5075.331} C_VEL
LIN {X 0,Y 516.881,Z 241.604,A -85,B 0,C 180,E1 -5077.945,E2 -5077.945} C_VEL
LIN {X 0,Y 516.868,Z 241.601,A -85,B 0,C 180,E1 -5080.746,E2 -5080.746} C_VEL
LIN {X 0,Y 516.86,Z 241.604,A -85,B 0,C 180,E1 -5082.837,E2 -5082.837} C_VEL
LIN {X 0,Y 516.892,Z 241.8,A -85,B 0,C 180,E1 -5083.905,E2 -5083.905} C_VEL
LIN {X 0,Y 517.306,Z 244.709,A -85,B 0,C 180,E1 -5086.143,E2 -5086.143} C_VEL
LIN {X 0,Y 517.496,Z 247.774,A -85,B 0,C 180,E1 -5088.329,E2 -5088.329} C_VEL
LIN {X 0,Y 517.405,Z 251.405,A -85,B 0,C 180,E1 -5090.739,E2 -5090.739} C_VEL
LIN {X 0,Y 517.302,Z 255.49,A -85,B 0,C 180,E1 -5093.29,E2 -5093.29} C_VEL
LIN {X 0,Y 517.158,Z 260.335,A -85,B 0,C 180,E1 -5096.14,E2 -5096.14} C_VEL
LIN {X 0,Y 516.979,Z 265.351,A -85,B 0,C 180,E1 -5098.923,E2 -5098.923} C_VEL
LIN {X 0,Y 516.76,Z 271.421,A -85,B 0,C 180,E1 -5102.133,E2 -5102.133} C_VEL
LIN {X 0,Y 516.616,Z 277.2,A -85,B 0,C 180,E1 -5105.057,E2 -5105.057} C_VEL
LIN {X 0,Y 516.533,Z 282.629,A -85,B 0,C 180,E1 -5107.704,E2 -5107.704} C_VEL
LIN {X 0,Y 516.486,Z 287.704,A -85,B 0,C 180,E1 -5110.112,E2 -5110.112} C_VEL
LIN {X 0,Y 516.426,Z 293.038,A -85,B 0,C 180,E1 -5112.579,E2 -5112.579} C_VEL
LIN {X 0,Y 516.319,Z 300.187,A -85,B 0,C 180,E1 -5115.818,E2 -5115.818} C_VEL
LIN {X 0,Y 516.335,Z 300.99,A -85,B 0,C 180,E1 -5116.132,E2 -5116.132} C_VEL
LIN {X 0,Y 517.972,Z 311.142,A -85,B 0,C 180,E1 -5116.415,E2 -5116.415} C_VEL
LIN {X 0,Y 518.396,Z 316.322,A -85,B 0,C 180,E1 -5116.576,E2 -5116.576} C_VEL
LIN {X 0,Y 518.072,Z 328.606,A -85,B 0,C 180,E1 -5117.066,E2 -5117.066} C_VEL
LIN {X 0,Y 517.827,Z 339.036,A -85,B 0,C 180,E1 -5117.613,E2 -5117.613} C_VEL
LIN {X 0,Y 517.632,Z 347.179,A -85,B 0,C 180,E1 -5118.133,E2 -5118.133} C_VEL
LIN {X 0,Y 517.35,Z 356.354,A -85,B 0,C 180,E1 -5118.838,E2 -5118.838} C_VEL
LIN {X 0,Y 517.119,Z 364.887,A -85,B 0,C 180,E1 -5119.626,E2 -5119.626} C_VEL
LIN {X 0,Y 516.946,Z 372.109,A -85,B 0,C 180,E1 -5120.413,E2 -5120.413} C_VEL
LIN {X 0,Y 516.728,Z 378.31,A -85,B 0,C 180,E1 -5121.199,E2 -5121.199} C_VEL
LIN {X 0,Y 516.591,Z 384.848,A -85,B 0,C 180,E1 -5122.181,E2 -5122.181} C_VEL
LIN {X 0,Y 516.477,Z 390.548,A -85,B 0,C 180,E1 -5123.212,E2 -5123.212} C_VEL
LIN {X 0,Y 516.419,Z 394.838,A -85,B 0,C 180,E1 -5124.142,E2 -5124.142} C_VEL
LIN {X 0,Y 516.277,Z 399.156,A -85,B 0,C 180,E1 -5125.315,E2 -5125.315} C_VEL
LIN {X 0,Y 516.355,Z 401.522,A -85,B 0,C 180,E1 -5126.098,E2 -5126.098} C_VEL
LIN {X 0,Y 516.285,Z 403.315,A -85,B 0,C 180,E1 -5126.879,E2 -5126.879} C_VEL
LIN {X 0,Y 516.193,Z 405.753,A -85,B 0,C 180,E1 -5128.44,E2 -5128.44} C_VEL
LIN {X 0,Y 516.161,Z 406.339,A -85,B 0,C 180,E1 -5129.22,E2 -5129.22} C_VEL
LIN {X 0,Y 516.161,Z 406.339,A -85,B 0,C 180,E1 -5130.78,E2 -5130.78} C_VEL
LIN {X 0,Y 516.193,Z 405.753,A -85,B 0,C 180,E1 -5131.56,E2 -5131.56} C_VEL
LIN {X 0,Y 516.285,Z 403.315,A -85,B 0,C 180,E1 -5133.121,E2 -5133.121} C_VEL
LIN {X 0,Y 516.316,Z 400.372,A -85,B 0,C 180,E1 -5134.293,E2 -5134.293} C_VEL
LIN {X 0,Y 516.375,Z 396.39,A -85,B 0,C 180,E1 -5135.467,E2 -5135.467} C_VEL
LIN {X 0,Y 516.434,Z 391.667,A -85,B 0,C 180,E1 -5136.56,E2 -5136.56} C_VEL
LIN {X 0,Y 516.55,Z 386.003,A -85,B 0,C 180,E1 -5137.623,E2 -5137.623} C_VEL
LIN {X 0,Y 516.718,Z 379.687,A -85,B 0,C 180,E1 -5138.604,E2 -5138.604} C_VEL
LIN {X 0,Y 516.894,Z 373.736,A -85,B 0,C 180,E1 -5139.39,E2 -5139.39} C_VEL
LIN {X 0,Y 517.045,Z 366.806,A -85,B 0,C 180,E1 -5140.178,E2 -5140.178} C_VEL
LIN {X 0,Y 517.318,Z 358.625,A -85,B 0,C 180,E1 -5140.964,E2 -5140.964} C_VEL
LIN {X 0,Y 517.552,Z 350.111,A -85,B 0,C 180,E1 -5141.653,E2 -5141.653} C_VEL
LIN {X 0,Y 517.695,Z 341.588,A -85,B 0,C 180,E1 -5142.234,E2 -5142.234} C_VEL
LIN {X 0,Y 518.029,Z 331.63,A -85,B 0,C 180,E1 -5142.786,E2 -5142.786} C_VEL
LIN {X 0,Y 518.224,Z 322.833,A -85,B 0,C 180,E1 -5143.179,E2 -5143.179} C_VEL
LIN {X 0,Y 518.33,Z 313.339,A -85,B 0,C 180,E1 -5143.513,E2 -5143.513} C_VEL
LIN {X 0,Y 516.473,Z 302.296,A -85,B 0,C 180,E1 -5143.839,E2 -5143.839} C_VEL
LIN {X 0,Y 516.317,Z 300.867,A -85,B 0,C 180,E1 -5143.881,E2 -5143.881} C_VEL
LIN {X 0,Y 516.348,Z 294.807,A -85,B 0,C 180,E1 -5146.608,E2 -5146.608} C_VEL
LIN {X 0,Y 516.443,Z 289.468,A -85,B 0,C 180,E1 -5149.062,E2 -5149.062} C_VEL
LIN {X 0,Y 516.5,Z 284.167,A -85,B 0,C 180,E1 -5151.554,E2 -5151.554} C_VEL
LIN {X 0,Y 516.618,Z 278.512,A -85,B 0,C 180,E1 -5154.289,E2 -5154.289} C_VEL
LIN {X 0,Y 516.751,Z 272.027,A -85,B 0,C 180,E1 -5157.542,E2 -5157.542} C_VEL
LIN {X 0,Y 516.898,Z 266.935,A -85,B 0,C 180,E1 -5160.203,E2 -5160.203} C_VEL
LIN {X 0,Y 517.074,Z 261.972,A -85,B 0,C 180,E1 -5162.933,E2 -5162.933} C_VEL
LIN {X 0,Y 517.233,Z 257.066,A -85,B 0,C 180,E1 -5165.75,E2 -5165.75} C_VEL
LIN {X 0,Y 517.367,Z 252.321,A -85,B 0,C 180,E1 -5168.672,E2 -5168.672} C_VEL
LIN {X 0,Y 517.491,Z 249.214,A -85,B 0,C 180,E1 -5170.683,E2 -5170.683} C_VEL
LIN {X 0,Y 517.457,Z 246.109,A -85,B 0,C 180,E1 -5172.823,E2 -5172.823} C_VEL
LIN {X 0,Y 517.084,Z 243.163,A -85,B 0,C 180,E1 -5175.025,E2 -5175.025} C_VEL
LIN {X 0,Y 516.889,Z 241.782,A -85,B 0,C 180,E1 -5176.105,E2 -5176.105} C_VEL
LIN {X 0,Y 516.906,Z 241.6,A -85,B 0,C 180,E1 -5178.398,E2 -5178.398} C_VEL
LIN {X 0,Y 516.879,Z 241.598,A -85,B 0,C 180,E1 -5181.281,E2 -5181.281} C_VEL
LIN {X 0,Y 516.869,Z 241.606,A -85,B 0,C 180,E1 -5184.216,E2 -5184.216} C_VEL
LIN {X 0,Y 516.891,Z 241.594,A -85,B 0,C 180,E1 -5187.05,E2 -5187.05} C_VEL
LIN {X 0,Y 516.885,Z 241.601,A -85,B 0,C 180,E1 -5189.793,E2 -5189.793} C_VEL
LIN {X 0,Y 516.878,Z 241.597,A -85,B 0,C 180,E1 -5192.461,E2 -5192.461} C_VEL
LIN {X 0,Y 516.861,Z 241.598,A -85,B 0,C 180,E1 -5195.066,E2 -5195.066} C_VEL
LIN {X 0,Y 516.87,Z 241.603,A -85,B 0,C 180,E1 -5197.618,E2 -5197.618} C_VEL
LIN {X 0,Y 516.928,Z 241.593,A -85,B 0,C 180,E1 -5200.126,E2 -5200.126} C_VEL
LIN {X 0,Y 516.893,Z 241.594,A -85,B 0,C 180,E1 -5202.591,E2 -5202.591} C_VEL
LIN {X 0,Y 516.939,Z 241.589,A -85,B 0,C 180,E1 -5205.026,E2 -5205.026} C_VEL
LIN {X 0,Y 516.962,Z 241.586,A -85,B 0,C 180,E1 -5208.23,E2 -5208.23} C_VEL
LIN {X 0,Y 516.923,Z 241.598,A -85,B 0,C 180,E1 -5211.395,E2 -5211.395} C_VEL
LIN {X 0,Y 516.978,Z 241.587,A -85,B 0,C 180,E1 -5213.752,E2 -5213.752} C_VEL
LIN {X 0,Y 516.963,Z 241.588,A -85,B 0,C 180,E1 -5216.878,E2 -5216.878} C_VEL
LIN {X 0,Y 517.083,Z 241.578,A -85,B 0,C 180,E1 -5219.217,E2 -5219.217} C_VEL
LIN {X 0,Y 517.063,Z 241.573,A -85,B 0,C 180,E1 -5222.332,E2 -5222.332} C_VEL
LIN {X 0,Y 516.999,Z 241.584,A -85,B 0,C 180,E1 -5225.455,E2 -5225.455} C_VEL
LIN {X 0,Y 516.944,Z 241.588,A -85,B 0,C 180,E1 -5227.809,E2 -5227.809} C_VEL
LIN {X 0,Y 516.934,Z 241.598,A -85,B 0,C 180,E1 -5230.967,E2 -5230.967} C_VEL
LIN {X 0,Y 516.869,Z 241.597,A -85,B 0,C 180,E1 -5234.161,E2 -5234.161} C_VEL
LIN {X 0,Y 516.882,Z 241.6,A -85,B 0,C 180,E1 -5236.585,E2 -5236.585} C_VEL
LIN {X 0,Y 516.875,Z 241.601,A -85,B 0,C 180,E1 -5239.04,E2 -5239.04} C_VEL
LIN {X 0,Y 516.857,Z 241.598,A -85,B 0,C 180,E1 -5241.533,E2 -5241.533} C_VEL
LIN {X 0,Y 516.876,Z 241.6,A -85,B 0,C 180,E1 -5244.923,E2 -5244.923} C_VEL
LIN {X 0,Y 516.892,Z 241.595,A -85,B 0,C 180,E1 -5247.901,E2 -5247.901} C_VEL
LIN {X 0,Y 516.854,Z 241.603,A -85,B 0,C 180,E1 -5250.199,E2 -5250.199} C_VEL
LIN {X 0,Y 516.857,Z 241.6,A -85,B 0,C 180,E1 -5252.942,E2 -5252.942} C_VEL
LIN {X 0,Y 516.85,Z 241.601,A -85,B 0,C 180,E1 -5255.774,E2 -5255.774} C_VEL
LIN {X 0,Y 516.841,Z 241.603,A -85,B 0,C 180,E1 -5258.711,E2 -5258.711} C_VEL
LIN {X 0,Y 516.878,Z 241.598,A -85,B 0,C 180,E1 -5261.769,E2 -5261.769} C_VEL
LIN {X 0,Y 516.872,Z 241.596,A -85,B 0,C 180,E1 -5265.006,E2 -5265.006} C_VEL
LIN {X 0,Y 516.876,Z 241.599,A -85,B 0,C 180,E1 -5268.393,E2 -5268.393} C_VEL
LIN {X 0,Y 516.881,Z 241.6,A -85,B 0,C 180,E1 -5270.274,E2 -5270.274} C_VEL
LIN {X 0,Y 516.246,Z 241.684,A -85,B 0,C 180,E1 -5270.924,E2 -5270.924} C_VEL
LIN {X 0,Y 513.382,Z 242.045,A -85,B 0,C 180,E1 -5271.979,E2 -5271.979} C_VEL
LIN {X 0,Y 510.93,Z 242.348,A -85,B 0,C 180,E1 -5272.828,E2 -5272.828} C_VEL
LIN {X 0,Y 509.867,Z 242.475,A -85,B 0,C 180,E1 -5273.485,E2 -5273.485} C_VEL
LIN {X 0,Y 509.776,Z 242.485,A -85,B 0,C 180,E1 -5273.707,E2 -5273.707} C_VEL
LIN {X 0,Y 509.805,Z 242.477,A -85,B 0,C 180,E1 -5276.536,E2 -5276.536} C_VEL
LIN {X 0,Y 509.791,Z 242.481,A -85,B 0,C 180,E1 -5279.331,E2 -5279.331} C_VEL
LIN {X 0,Y 509.835,Z 242.477,A -85,B 0,C 180,E1 -5282.052,E2 -5282.052} C_VEL
LIN {X 0,Y 509.836,Z 242.473,A -85,B 0,C 180,E1 -5284.702,E2 -5284.702} C_VEL
LIN {X 0,Y 509.819,Z 242.482,A -85,B 0,C 180,E1 -5287.44,E2 -5287.44} C_VEL
LIN {X 0,Y 509.851,Z 242.476,A -85,B 0,C 180,E1 -5289.843,E2 -5289.843} C_VEL
LIN {X 0,Y 509.838,Z 242.48,A -85,B 0,C 180,E1 -5293.174,E2 -5293.174} C_VEL
LIN {X 0,Y 509.816,Z 242.482,A -85,B 0,C 180,E1 -5295.633,E2 -5295.633} C_VEL
LIN {X 0,Y 509.875,Z 242.47,A -85,B 0,C 180,E1 -5298.1,E2 -5298.1} C_VEL
LIN {X 0,Y 509.884,Z 242.475,A -85,B 0,C 180,E1 -5301.279,E2 -5301.279} C_VEL
LIN {X 0,Y 509.924,Z 242.466,A -85,B 0,C 180,E1 -5303.67,E2 -5303.67} C_VEL
LIN {X 0,Y 509.922,Z 242.47,A -85,B 0,C 180,E1 -5306.84,E2 -5306.84} C_VEL
LIN {X 0,Y 509.983,Z 242.457,A -85,B 0,C 180,E1 -5310,E2 -5310} C_VEL
LIN {X 0,Y 509.922,Z 242.47,A -85,B 0,C 180,E1 -5313.16,E2 -5313.16} C_VEL
LIN {X 0,Y 509.924,Z 242.466,A -85,B 0,C 180,E1 -5316.33,E2 -5316.33} C_VEL
LIN {X 0,Y 509.884,Z 242.475,A -85,B 0,C 180,E1 -5318.721,E2 -5318.721} C_VEL
LIN {X 0,Y 509.883,Z 242.469,A -85,B 0,C 180,E1 -5321.932,E2 -5321.932} C_VEL
LIN {X 0,Y 509.856,Z 242.474,A -85,B 0,C 180,E1 -5325.256,E2 -5325.256} C_VEL
LIN {X 0,Y 509.844,Z 242.476,A -85,B 0,C 180,E1 -5328.011,E2 -5328.011} C_VEL
LIN {X 0,Y 509.796,Z 242.48,A -85,B 0,C 180,E1 -5331.003,E2 -5331.003} C_VEL
LIN {X 0,Y 509.805,Z 242.477,A -85,B 0,C 180,E1 -5333.564,E2 -5333.564} C_VEL
LIN {X 0,Y 509.854,Z 242.479,A -85,B 0,C 180,E1 -5336.383,E2 -5336.383} C_VEL
LIN {X 0,Y 509.829,Z 242.475,A -85,B 0,C 180,E1 -5338.846,E2 -5338.846} C_VEL
LIN {X 0,Y 509.767,Z 242.483,A -85,B 0,C 180,E1 -5341.593,E2 -5341.593} C_VEL
LIN {X 0,Y 509.797,Z 242.482,A -85,B 0,C 180,E1 -5344.417,E2 -5344.417} C_VEL
LIN {X 0,Y 509.765,Z 242.482,A -85,B 0,C 180,E1 -5347.344,E2 -5347.344} C_VEL
LIN {X 0,Y 509.83,Z 242.477,A -85,B 0,C 180,E1 -5350.382,E2 -5350.382} C_VEL
LIN {X 0,Y 509.789,Z 242.479,A -85,B 0,C 180,E1 -5353.069,E2 -5353.069} C_VEL
LIN {X 0,Y 509.813,Z 242.483,A -85,B 0,C 180,E1 -5355.793,E2 -5355.793} C_VEL
LIN {X 0,Y 509.824,Z 242.475,A -85,B 0,C 180,E1 -5358.581,E2 -5358.581} C_VEL
LIN {X 0,Y 509.808,Z 242.484,A -85,B 0,C 180,E1 -5361.791,E2 -5361.791} C_VEL
LIN {X 0,Y 509.805,Z 242.476,A -85,B 0,C 180,E1 -5364.628,E2 -5364.628} C_VEL
LIN {X 0,Y 509.824,Z 242.482,A -85,B 0,C 180,E1 -5367.486,E2 -5367.486} C_VEL
LIN {X 0,Y 509.822,Z 242.475,A -85,B 0,C 180,E1 -5370.279,E2 -5370.279} C_VEL
LIN {X 0,Y 509.851,Z 242.473,A -85,B 0,C 180,E1 -5372.949,E2 -5372.949} C_VEL
LIN {X 0,Y 509.832,Z 242.479,A -85,B 0,C 180,E1 -5375.579,E2 -5375.579} C_VEL
LIN {X 0,Y 509.822,Z 242.479,A -85,B 0,C 180,E1 -5379.003,E2 -5379.003} C_VEL
LIN {X 0,Y 509.835,Z 242.477,A -85,B 0,C 180,E1 -5381.521,E2 -5381.521} C_VEL
LIN {X 0,Y 509.887,Z 242.471,A -85,B 0,C 180,E1 -5384.824,E2 -5384.824} C_VEL
LIN {X 0,Y 509.884,Z 242.467,A -85,B 0,C 180,E1 -5388.127,E2 -5388.127} C_VEL
LIN {X 0,Y 509.884,Z 242.471,A -85,B 0,C 180,E1 -5391.284,E2 -5391.284} C_VEL
LIN {X 0,Y 509.922,Z 242.462,A -85,B 0,C 180,E1 -5393.675,E2 -5393.675} C_VEL
LIN {X 0,Y 509.938,Z 242.469,A -85,B 0,C 180,E1 -5396.845,E2 -5396.845} C_VEL
LIN {X 0,Y 510.049,Z 242.449,A -85,B 0,C 180,E1 -5399.215,E2 -5399.215} C_VEL
LIN {X 0,Y 509.913,Z 242.463,A -85,B 0,C 180,E1 -5401.584,E2 -5401.584} C_VEL
LIN {X 0,Y 509.906,Z 242.466,A -85,B 0,C 180,E1 -5403.165,E2 -5403.165} C_VEL
LIN {X 0,Y 509.932,Z 242.466,A -85,B 0,C 180,E1 -5406.334,E2 -5406.334} C_VEL
LIN {X 0,Y 509.878,Z 242.474,A -85,B 0,C 180,E1 -5408.725,E2 -5408.725} C_VEL
LIN {X 0,Y 509.9,Z 242.467,A -85,B 0,C 180,E1 -5411.936,E2 -5411.936} C_VEL
LIN {X 0,Y 509.892,Z 242.466,A -85,B 0,C 180,E1 -5415.246,E2 -5415.246} C_VEL
LIN {X 0,Y 509.855,Z 242.476,A -85,B 0,C 180,E1 -5418.488,E2 -5418.488} C_VEL
LIN {X 0,Y 509.849,Z 242.471,A -85,B 0,C 180,E1 -5421.005,E2 -5421.005} C_VEL
LIN {X 0,Y 509.821,Z 242.476,A -85,B 0,C 180,E1 -5423.567,E2 -5423.567} C_VEL
LIN {X 0,Y 509.846,Z 242.476,A -85,B 0,C 180,E1 -5426.366,E2 -5426.366} C_VEL
LIN {X 0,Y 509.85,Z 242.471,A -85,B 0,C 180,E1 -5428.849,E2 -5428.849} C_VEL
LIN {X 0,Y 509.821,Z 242.478,A -85,B 0,C 180,E1 -5431.593,E2 -5431.593} C_VEL
LIN {X 0,Y 509.842,Z 242.474,A -85,B 0,C 180,E1 -5434.417,E2 -5434.417} C_VEL
LIN {X 0,Y 509.811,Z 242.48,A -85,B 0,C 180,E1 -5437.344,E2 -5437.344} C_VEL
LIN {X 0,Y 509.823,Z 242.48,A -85,B 0,C 180,E1 -5440.387,E2 -5440.387} C_VEL
LIN {X 0,Y 509.806,Z 242.484,A -85,B 0,C 180,E1 -5443.062,E2 -5443.062} C_VEL
LIN {X 0,Y 509.817,Z 242.609,A -85,B 0,C 180,E1 -5443.575,E2 -5443.575} C_VEL
LIN {X 0,Y 510.345,Z 246.342,A -85,B 0,C 180,E1 -5446.486,E2 -5446.486} C_VEL
LIN {X 0,Y 510.478,Z 250.214,A -85,B 0,C 180,E1 -5449.222,E2 -5449.222} C_VEL
LIN {X 0,Y 510.345,Z 254.015,A -85,B 0,C 180,E1 -5451.719,E2 -5451.719} C_VEL
LIN {X 0,Y 510.197,Z 258.782,A -85,B 0,C 180,E1 -5454.652,E2 -5454.652} C_VEL
LIN {X 0,Y 510.012,Z 263.666,A -85,B 0,C 180,E1 -5457.493,E2 -5457.493} C_VEL
LIN {X 0,Y 509.833,Z 268.718,A -85,B 0,C 180,E1 -5460.282,E2 -5460.282} C_VEL
LIN {X 0,Y 509.672,Z 273.739,A -85,B 0,C 180,E1 -5462.933,E2 -5462.933} C_VEL
LIN {X 0,Y 509.563,Z 278.883,A -85,B 0,C 180,E1 -5465.559,E2 -5465.559} C_VEL
LIN {X 0,Y 509.429,Z 284.099,A -85,B 0,C 180,E1 -5468.131,E2 -5468.131} C_VEL
LIN {X 0,Y 509.363,Z 289.37,A -85,B 0,C 180,E1 -5470.662,E2 -5470.662} C_VEL
LIN {X 0,Y 509.293,Z 294.68,A -85,B 0,C 180,E1 -5473.155,E2 -5473.155} C_VEL
LIN {X 0,Y 509.248,Z 300.709,A -85,B 0,C 180,E1 -5475.923,E2 -5475.923} C_VEL
LIN {X 0,Y 511.253,Z 313.14,A -85,B 0,C 180,E1 -5476.296,E2 -5476.296} C_VEL
LIN {X 0,Y 511.377,Z 318.774,A -85,B 0,C 180,E1 -5476.489,E2 -5476.489} C_VEL
LIN {X 0,Y 511.122,Z 329.419,A -85,B 0,C 180,E1 -5476.938,E2 -5476.938} C_VEL
LIN {X 0,Y 510.856,Z 338.88,A -85,B 0,C 180,E1 -5477.444,E2 -5477.444} C_VEL
LIN {X 0,Y 510.638,Z 347.428,A -85,B 0,C 180,E1 -5478.002,E2 -5478.002} C_VEL
LIN {X 0,Y 510.361,Z 356.159,A -85,B 0,C 180,E1 -5478.684,E2 -5478.684} C_VEL
LIN {X 0,Y 510.084,Z 364.691,A -85,B 0,C 180,E1 -5479.481,E2 -5479.481} C_VEL
LIN {X 0,Y 509.912,Z 371.913,A -85,B 0,C 180,E1 -5480.28,E2 -5480.28} C_VEL
LIN {X 0,Y 509.686,Z 378.115,A -85,B 0,C 180,E1 -5481.076,E2 -5481.076} C_VEL
LIN {X 0,Y 509.522,Z 384.652,A -85,B 0,C 180,E1 -5482.072,E2 -5482.072} C_VEL
LIN {X 0,Y 509.413,Z 390.207,A -85,B 0,C 180,E1 -5483.087,E2 -5483.087} C_VEL
LIN {X 0,Y 509.316,Z 394.642,A -85,B 0,C 180,E1 -5484.06,E2 -5484.06} C_VEL
LIN {X 0,Y 509.194,Z 398.961,A -85,B 0,C 180,E1 -5485.25,E2 -5485.25} C_VEL
LIN {X 0,Y 509.248,Z 401.326,A -85,B 0,C 180,E1 -5486.043,E2 -5486.043} C_VEL
LIN {X 0,Y 509.203,Z 403.121,A -85,B 0,C 180,E1 -5486.835,E2 -5486.835} C_VEL
